METHOD Init
VAR_INPUT
  pMsgConfig : POINTER TO ST_MSG_CONFIG;         // message config
  fPrintResolution : LREAL := 1;                 // print(head) resolution in [dpi]
  fSubPxResolution : LREAL := 1;                 // SubPixel resolution [SubPx], resolution factor (fI_PrintResolution*fI_SubPxResolution=>Output resolution)
  bParallelCT : BOOL;                            // Support parallel processing of CTs
END_VAR
SUPER^.Init(pMsgConfig:=pMsgConfig, fPrintResolution:=fPrintResolution, fSubPxResolution:=fSubPxResolution, bParallelCT:=bParallelCT);

// Init messages
fbMsg_PythonNotRunning.pI_MsgConfig := _pMsgConfigExt;
fbMsg_PythonNotRunning.iI_MsgLocation := TO_INT(ePr_BLK_PU);
fbMsg_PythonNotRunning.iI_MsgNumber := eC_STAG_DEF_SCRIPT_NOT_RUNNING;
END_METHOD

METHOD InitWorkerPython
VAR_INPUT
  aScriptPath : T_MaxString;                     // path to cmd scripts
  //aAmsLocalHost : T_AmsNetID;                    // Ams netId localhost of the pc to run the script
  iDefGridParamMediator : I_ParamMediator;
END_VAR
IF NOT bInitialized OR _pCTM = 0 THEN LogError('Base Worker not initialized! call init() before'); RETURN; END_IF
IF iDefGridParamMediator = 0 THEN bInitialized := FALSE; LogError('Invalid parameter, no valid param mediator'); RETURN; END_IF

// worker specific init
_iParamMediator := iDefGridParamMediator;

fbPythonInterface.Init(
  sCTManagerPath := _pCTM^.sCTDefGridInstancesPath, 
  sScriptPath:=aScriptPath
);
END_METHOD

METHOD mJobStart
VAR_INPUT
	sJobDef	: CalmarCompPrint.I_JobDefinition;
END_VAR
// checks and fix defaults
IF _iParamMediator = 0 THEN LogError('JobStart: invalid parameter configuration'); RETURN; END_IF
IF _fWorkerPosition = 0 THEN _fWorkerPosition := fC_DEFAULT_WOKER_POSITION; LogError(F_Concat3(_name, ': worker position not set, set default=', TO_STRING(fC_DEFAULT_WOKER_POSITION))); END_IF

// configure
_aJobName := sJobDef.aJobName;
_aJobGuid := sJobDef.aJobId;
_fImageDepthM := sJobDef.fImageDepth/1000;
_fImageWidthM := sJobDef.fImageWidth/1000;

_bNewJob := TRUE;
_bJobActive := TRUE;
END_METHOD

METHOD  mJobStop
VAR_INPUT
	sStatus	: CalmarCompPrint.I_JobStatus;
END_VAR
fbPythonInterface.JobStop();
_bJobActive := FALSE;
END_METHOD

METHOD  work
VAR_INPUT
END_VAR
VAR
  i : UDINT;
  tempCt  : POINTER TO FB_ContainerDefGrid;
  bDeformationDone : BOOL;
  bDeformationError : BOOL;
END_VAR
VAR_INST
  rT_EnablePyIf  : R_TRIG;
END_VAR
SUPER^.work();

IF _iParamMediator = 0 THEN F_Report_Error(ErrType:=EN_REPORT_ERROR_TYPE.Report_Error_0Pointer); RETURN; END_IF
_CamGridSettings := _iParamMediator.sCameraGridSettings;
_DefGridSettings := _iParamMediator.sDeformationGridSettings;

// reconfig script after job started (Mediator parameter are defined in JobStart())
IF _bNewJob OR rT_EnablePyIf.Q THEN   // new job activated or re-enabled
  _bNewJob := FALSE;
  
  // setup script
  fbPythonInterface.JobStart(
    aJobName:=_aJobName,
    aJobGuid:=_aJobGuid,
    nJobImageWidth:=DINT_TO_UDINT(F_MeterToSubPixel(fPosMeter:=_fImageDepthM, fResoSubPx:=_fPrintResolution)),
    nJobImageHeigth:=DINT_TO_UDINT(F_MeterToSubPixel(fPosMeter:=_fImageWidthM, fResoSubPx:=_fPrintResolution)),
    nCamFrameWidth:=DINT_TO_UDINT(FC_LREAL_TO_DINT(_CamGridSettings.fGridFeaturePitch)),
    pGridSettings:=ADR(_DefGridSettings)
  );
END_IF

// start/stop script
IF _CamGridSettings.eCameraMode >= E_CameraMode.Live AND THIS^.bWorkerEnable THEN 
  fbPythonInterface.bEnable := TRUE;
ELSE
  fbPythonInterface.bEnable := FALSE;
END_IF
rT_EnablePyIf(CLK:=fbPythonInterface.bEnable);

fbPythonInterface();

IF _pAttachedCt <> 0 THEN
  // nothing to do anymore just release CT
  // NOTE: the delete of the CT is done by DeleteDefCt() method directly into fbPythonInterface
  Release(_pAttachedCt^);
END_IF

// messages
fbMsg_PythonNotRunning(bI_Status:=fbPythonInterface.bError);
IF fbMsg_PythonNotRunning.bMsgAck THEN fbPythonInterface.ackError(); END_IF
END_METHOD

END_FUNCTION_BLOCK

// ---- POUs/Print/DefGrid/FB_WorkerDefGrid_Verify.TcPOU
FUNCTION_BLOCK FB_WorkerDefGrid_Verify EXTENDS FB_WorkerDefGrid
VAR_OUTPUT
  bWateGateActive   AT%Q* : BOOL;     //  wate gate activation pulse
END_VAR
VAR
  bLastEject   : BOOL;   // stores state if last CT TRUE:=Eject, FALSE:=OK
  tpEjectPulse  : TP := (PT:=T#80MS);
  
  // print manager reference
  _pPm : POINTER TO FB_ProdManager_DMAX;
  
  // view verify history
  tpShowResult : TP := (PT:=T#700MS);
  nStateHistory : ARRAY[1..20] OF UINT;   // 2=???, 1=Eject, 0=OK
  nStateHistory_FillColor : ARRAY[1..20] OF UDINT;
  sResultText : STRING;
  
  // Grid Table export
  nCTId : DINT;
  bEnableGridExport : BOOL;
  nExportWrites : UDINT;
  sOutputPath : T_MaxString := 'C:\GridExport';
  sFileFormat : STRING := 'json';
  fbGridExporter : FB_GridDataExporter;
END_VAR

METHOD PROTECTED  Attach : BOOL
VAR_INPUT
  iCT              : I_CT;                         (*container at triggered event position*)
END_VAR
VAR 
  bSuccess         : BOOL;
END_VAR
IF SUPER^.Attach(iCT:=iCT) THEN
  
  // do CT supervision here and decice what happens with this sheet
   bSuccess := TRUE;
  IF NOT iCT.bValid AND iCT.bProductPresent AND iCT.pJob <> 0 THEN
    bSuccess := FALSE;
    // tag for ejection
    iCT.pCT^.lPrOutput := EN_PrinterOutput.trash;
	END_IF

  // finish CT in production
  IF _pPm <> 0 THEN 
    _pPm^.CT_Finish(sCT:=iCT, bSuccess:=bSuccess);      // report to job status
  ELSE
    LogError('PrintManager not set');
	END_IF
  
  // select output
  IF iCT.pCT^.lPrOutput = EN_PrinterOutput.trash THEN
    // create eject trigger
    tpEjectPulse(IN:=TRUE);
    bLastEject := TRUE;
    LogLvl(Lvl:=E_LogSeverity.Debug, Msg:=F_Concat2('Eject CT: ', _pAttachedCt^.print(0)));
  ELSE
    tpEjectPulse(IN:=FALSE);
    bLastEject := FALSE;
	END_IF
  
  // History view
  MEMMOVE(destAddr:=ADR(nStateHistory[1+1]),           srcAddr:=ADR(nStateHistory[1]),           n:=((SIZEOF(nStateHistory)/SIZEOF(nStateHistory[1]))-1)*SIZEOF(nStateHistory[1]));
  MEMMOVE(destAddr:=ADR(nStateHistory_FillColor[1+1]), srcAddr:=ADR(nStateHistory_FillColor[1]), n:=((SIZEOF(nStateHistory_FillColor)/SIZEOF(nStateHistory_FillColor[1]))-1)*SIZEOF(nStateHistory_FillColor[1]));
  
  nStateHistory[1] := SEL(bLastEject=TRUE, 0, 1);
  sResultText := SEL(bLastEject=TRUE, 'OK', 'NOK');

  IF iCT.bProductPresent AND iCT.bValid THEN        nStateHistory_FillColor[1] := 16#FF000000 OR WebColors.LightGreen.lCode;
  ELSIF iCT.bProductPresent AND NOT iCT.bValid AND iCT.pCT^.lPrOutput = EN_PrinterOutput.trash THEN nStateHistory_FillColor[1] := 16#FF000000 OR WebColors.LightSalmon.lCode;   
  ELSIF iCT.bProductPresent AND NOT iCT.bValid AND iCT.pCT^.lPrOutput <> EN_PrinterOutput.trash THEN nStateHistory_FillColor[1] := 16#FF000000 OR WebColors.LightGray.lCode;
	ELSIF NOT iCT.bProductPresent THEN                nStateHistory_FillColor[1] := 16#FF000000 OR WebColors.LightGray.lCode;
  END_IF

  tpShowResult(IN:=FALSE);
  tpShowResult(IN:=TRUE);
  
  // grid history
  IF bEnableGridExport AND iCT.bProductPresent AND nExportWrites < 100 THEN
    nCTId := _pAttachedCt^.pCT^.iId;
    sFileFormat := SEL(sFileFormat='csv', 'json', 'csv');
    fbGridExporter(
        sOutputDir:=sOutputPath,
        sFileName:=F_Concat4('\Export_', TO_STRING(nCTId), '.', sFileFormat),
        pFbImageDeformation:=_pAttachedCt^.pImageDeformation,
        //nSelectGrid:=
    );
    fbGridExporter.startExport();
    nExportWrites:=nExportWrites+1;
  ELSE
    nExportWrites := 0; bEnableGridExport := FALSE;
  END_IF
END_IF
END_METHOD

(*
  Set PrintManager.
*)
METHOD InitWorkerVerify : BOOL
VAR_INPUT
  pPm : POINTER TO FB_ProdManager_DMAX;
END_VAR
IF pPm = 0 THEN LogError('Invalid Pm given'); END_IF

_pPm := pPm;  // register print manager reference
END_METHOD

METHOD   mJobStart
VAR_INPUT
	sJobDef	: CalmarCompPrint.I_JobDefinition;
END_VAR
END_METHOD

METHOD  mJobStop
VAR_INPUT
	sStatus	: CalmarCompPrint.I_JobStatus;
END_VAR
END_METHOD

METHOD Release : BOOL
VAR_INPUT
  iCT              : I_CT;                         (*container at triggered event position*)
END_VAR
IF SUPER^.Release(iCT := iCT) THEN
  ;
END_IF
END_METHOD

METHOD  work
VAR_INST
  fT_Pulse  : F_TRIG;
END_VAR
SUPER^.work();

// output signal handling
tpEjectPulse(Q=>bWateGateActive);
fT_Pulse(CLK:=bWateGateActive);
tpShowResult();
//IF tpShowResult.IN:=TRUE AND NOT tpShowResult.Q THEN tpShowResult(IN:=FALSE); END_IF   // reset pulse

fbGridExporter();

// release
IF tpEjectPulse.IN THEN
  IF fT_Pulse.Q THEN  
    tpEjectPulse(IN:=FALSE);
  END_IF
END_IF

IF _pAttachedCt <> 0 THEN   // just release any attached container in this cycle
  Release(iCT:=_pAttachedCt^);
END_IF
END_METHOD

END_FUNCTION_BLOCK

// ---- POUs/Print/Maxliner/FB_PrintModule_Maxliner.TcPOU
(*
  A DVT PrintModule (DEU, DSU, WEU).
*)
FUNCTION_BLOCK FB_PrintModule_Maxliner EXTENDS T_NamedBase IMPLEMENTS I_Sim, I_PositionEvent
VAR_INPUT
  // encoder input --> directly mapped into FB_PrintPosition 
  // machine state by pointer in init()
  // external start pos interface by pointer in init()
  fPrintOffsetX           : LREAL;   // [m] external configurative offsets to PM (PU)
  fPrintOffsetY           : LREAL;   // [m] external configurative offsets to PM (PU)

  fPUPlate1_Temperature   : LREAL;  // PU Plate1 temperature
END_VAR

VAR
  //config

  // - references
  _pModuleSetup           : POINTER TO ST_CassetteSetup;
  _iPrintGlobal           : I_PrintGlobal;        // master module (setting, position, global stuff, ...)
  _iPrintPosition         : I_PrintPosition;      // module's position
  _iStartPos              : I_StartPosDetect;     // module's start position detect
  _iModule                : I_Module;             // module's system status
  _pModuleMachineState    : POINTER TO ST_ModuleMachineInterface_IN;   // machine interface-print states
  _pModuleMachineFeedback : POINTER TO ST_ModuleMachineInterface_OUT;  // machine interface-print feedback
    
  // status
  bInit                   : BOOL;   // initialized
  bSelectedForPrint       : BOOL;   // selected for printing
  bReadyForPrinting       : BOOL;   // Module ready for printing
  bHardwareHold           : BOOL;   // hw hold
  _bGridLimited           : BOOL;   // calculated grid was limited before sending
  
  // instances
  fbPrintPosition         : FB_PrintPositionDmax;   // a position per pm (external encoder wheel)

  fbCTTracker             : FB_CTTracker;
  fbParamMediator         : FB_DefGridParamMediator;
  fbWorkerPython          : FB_WorkerDefGrid_Python;
  fbWorkerCamera          : FB_WorkerDefGrid_Camera;
  fbWorkerDeformation     : FB_WorkerDefGrid_Deformation;
  fbWorkerPrint           : ARRAY[1..GVL_Maxliner.nC_MaxWorkerPrintPerPm] OF FB_WorkerDefGrid_Print;
  
  _pAdsSa                 : POINTER TO FB_ADS_DVTSHEETALIGNMENT; // sheet alignement ads
  fbAdsPm                 : FB_ADS_PM;      // PM -  Print Module ADS
  fbAdsPg                 : ARRAY[1..GVL_Maxliner.nC_MaxWorkerPrintPerPm] OF FB_ADS_PG;  // PG - PrintGroup ADS
  
  // hw (references only for now) ------
  // - pc
  _pPc                    : ARRAY[1..GVL_Maxliner.nC_MaxPcPerPm] OF POINTER TO FB_PC;
  _nPc                    : UDINT;  // number of PC in module
  _nPcToWorker_Mapping    : ARRAY[1..GVL_Maxliner.nC_MaxPcPerPm] OF UDINT;   // Mapping of PC to worker  
  _nPcToPgAbsoluteIdx     : ARRAY[1..GVL_Maxliner.nC_MaxPcPerPm] OF UDINT;   // Mapping of PC to absolute PG index
  // - ph
  _pPh                    : ARRAY[1..GVL_Maxliner.nC_MaxPhPerPm] OF POINTER TO FB_PH;
  _nPh                    : UDINT;  // number of PH in module
  _nPhToWorker_Mapping    : ARRAY[1..GVL_Maxliner.nC_MaxPhPerPm] OF UDINT;  // Mapping of PH to worker
  _nPhToPc_Mapping        : ARRAY[1..GVL_Maxliner.nC_MaxPhPerPm] OF UDINT;  // Mapping of PH to PC
  _nPhToPcCh_Mapping      : ARRAY[1..GVL_Maxliner.nC_MaxPhPerPm] OF UDINT;  // Mapping of PH to PC channel
  _nPhToPgAbsoluteIdx     : ARRAY[1..GVL_Maxliner.nC_MaxPhPerPm] OF UDINT;  // Mapping of PH to absolute PG index
  
  // helper
  nCtr                    : UDINT;
  nYShift_PcRamCenter     : UDINT;     // y-shift for centered image in CB RAM [px]
  fSpeed, fSpeedMpMin     : LREAL;
  bSpeedReachedForPrinting: BOOL;      // Speed for printing reached
  nPos_SubPx, nPos_Px     : DINT;
  nPos_SubPx_mem          : DINT;
  fPos_um                 : LREAL;
  nTrackPosMain           : DINT;      // tracker attach position - module position relative to pos reference in main tracker [m]

  bHwSyncCmd              : BOOL;
  sCamGridSettings        : ST_CameraGridSettings;
  bOnePgActive            : BOOL;

  // sync CT trigger with Camera detection
  _bNewCT                 : BOOL;   // a new ct is received to be treated
  _iNewCT                 : I_CT;   // new ct to be treated
  _bNewStartPosX0         : BOOL;   // a new startpos detected by cam
  _nNewStartPosX0         : DINT;   // new startpos X0 deteced by cam

  fbFineAlignement        : FB_FineAlignement;     // additional grid corrections, PU Deformation/correction (4p, banana, ...)

  // messaging
  fb_MsgQueue             : FB_MSG_QUEUE;                 (*Message queue*)
  fb_MsgHandler           : FB_MSG_HANDLER;               (*Message handler*)
  sL_MsgConfig            : ST_MSG_CONFIG;                (*Message config*)
//fbMsg                   : ARRAY [1..nC_NumMsg] OF FB_MESSAGE;  (*Messages*)
  
  // simulation
  fbSim                   : FB_Sim;

  // view
  fbView                  : FB_PrintModule_Maxliner_View;    // additional controls for print module visus

  // test
  bTestMsg : BOOL;      // activate message test
END_VAR

VAR PERSISTENT
  _fPmDistToPrev          : LREAL;                 // [m] distance to previous PM (in main domain)
  _fPmMainTrackPos        : LREAL;                 // [m] used distance to master reference position (in main tracker)
END_VAR

VAR CONSTANT
  nC_NumMsg               : UDINT := 0;            // number of internal messages
  fC_HeadOffsetPlate      : LREAL := 0.000_2;      // Head offset to base plate [m] (mechanical)
  fC_MinimalProductionSpeed_in_MpMin: LREAL := 5.0;    // [m/min]
  fC_FormatLengthTolerance : LREAL := 100.0;       // [px] tolerance of substrate length job - machine config 
  nC_StopReadyTimeout     : TIME := T#10S;         // Synced stopping of printing, max. timeout to wait for printing end
END_VAR

IF NOT bInit THEN RETURN; END_IF

// position
fbPrintPosition.fEnoderResolution := _pModuleMachineState^.fEncoderResolution;    // encoder resolution from machine
fbPrintPosition();

// -------------------------
// StartTrigger evaluation -> apply new CT to Tracking (created from CTM externally)
// Synchronize CT (EvPos) received from CTManger (Main) to the local StartTrigger detection and positioning
// -- reset triggers if not active
IF NOT bReadyForPrinting THEN
  _bNewCT := 0; _bNewStartPosX0 := 0;
END_IF
// -- new StartTrigger (X0)
IF bReadyForPrinting AND _iStartPos.bStartTrig AND _iStartPos.bValid THEN
  // buffer/save new start trigger
  _bNewStartPosX0 := TRUE;
  _nNewStartPosX0 := _iStartPos.nStartPositionX0;      // save detected start position for next CT to be applied to this module¨
  
  LogLvl(Lvl:=E_LogSeverity.Debug, Msg:=F_Concat3(
    F_Concat2(_pModuleSetup^.aName, ' New StartTrigger detected:'),
    F_Concat2(' at position X0:', TO_STRING(_nNewStartPosX0)),
    F_Concat2(' PM is now at: ', TO_STRING(fbPrintPosition.getPosition())),
  ));
  
  IF _bNewCT THEN   // we have an attached CT
      LogLvl(Lvl:=E_LogSeverity.Debug, Msg:=F_Concat3(
      F_Concat2(_pModuleSetup^.aName, ' Track NewCT:'),
      F_Concat2(' internal (print)Pos X0:', TO_STRING(_nNewStartPosX0)),
      F_Concat2(' with CT:', _iNewCT.print(0))
    ));
    
    _iNewCT.nPosPrint_X0 := _nNewStartPosX0;                            // set print pos to new dected in this module position domain
    fbCTTracker.RegisterCT(iCT := _iNewCT, nX0 := _nNewStartPosX0);     // register ct for tracking in modules position and tracking system
  ELSE
    // spurious trigger (CTs not yet arrived at PMx, but receive some StartTriggers
    LogLvl(Lvl:=E_LogSeverity.Debug, Msg:=F_Concat3('StartTrigger at Pos X0:', TO_STRING(_nNewStartPosX0), ' but no CT received'));
	END_IF
  
  // reset internals (saved triggers)
  _bNewCT := FALSE; _iNewCT := 0; 
  _bNewStartPosX0 := FALSE;
END_IF

// positioning
// - get position 
nPos_SubPx := _iPrintPosition.getPosition(nPosition_px=>nPos_Px, fPosition_um=>fPos_um);
// (disabled) nPos_SubPx := nPos_SubPx_mem := SEL(bReadyForPrinting AND _iPrintPosition.bMoving, nPos_SubPx_mem, nPos_SubPx);   // security measure (jetting when not really moving or not in position
// - get speed
fSpeed := _iPrintPosition.getSpeed(fSpeedMpMin=>fSpeedMpMin);

// update distance from machine
_fPmDistToPrev := _pModuleMachineState^.fDistanceToPrevModule;

// enable, control, release signals
//   engaged -> selected and prepared for production
//   printActivated -> machine & axis position ready for printing
//   InitInPrintPosition -> module in pos to allow printing
bSelectedForPrint        := fbAdsPm.bEnable AND _pModuleMachineState^.bEngaged;
bSpeedReachedForPrinting := (fSpeedMpMin >= fC_MinimalProductionSpeed_in_MpMin);
// ready for printing (enable detection)
bReadyForPrinting        :=      bSelectedForPrint                                // selected and ready for production (from machine)
                            AND _pModuleMachineState^.bPrintActivated             // machine & axis ready for printing
                            AND _pModuleMachineState^.bUnitInPrintPosition        // module in printing position -> allowed to print
                            AND bSpeedReachedForPrinting                          // speed bigger than min speed for printing
                            AND _pModuleMachineState^.bTargetSpeedReached         // do not evaluate marks while machine ramping up  
                            AND NOT _pModuleMachineState^.bStopRequest            // do not evaluate marks while machine is stopping
                            AND NOT _pModuleMachineState^.bEStop
                            AND NOT _pModuleMachineState^.bSleep;
bHardwareHold            := NOT bSpeedReachedForPrinting OR 
                            NOT _pModuleMachineState^.bPrintActivated OR 
                            NOT _pModuleMachineState^.bUnitInPrintPosition OR 
                                _pModuleMachineState^.bFastStopRequest;
bHwSyncCmd               := checkHwSyncRequest();                                 // sync trigger generation

// pos for attach in main tracker
nTrackPosMain := F_MeterToSubPixel(fPosMeter:=_fPmMainTrackPos, fResoSubPx:=_iPrintPosition.fPrintResolution*_iPrintPosition.fSubPxResolution); 
// run tracker
fbCTTracker(nPos:=nPos_SubPx);


// call hardware
(* -- PC PrintController*)
FOR nCtr := 1 TO _nPc DO
  IF _pPc[nCtr] <> 0 THEN
    _pPc[nCtr]^.sI_SystemCmd.bSleep := _pModuleMachineState^.bSleep;  // from if to module (machine)
    _pPc[nCtr]^.sI_SystemCmd.bEStop := _pModuleMachineState^.bEStop;  // from if to module (machine)
    _pPc[nCtr]^.sI_SystemCmd.bAirNotOk := FALSE;
    _pPc[nCtr]^();
  END_IF
END_FOR

(* -- PH PrintHead*)
FOR nCtr := 1 TO _nPh DO
  IF _pPh[nCtr] <> 0 THEN
    ; // called in PC.update()->pPh[nCtr]^();
  END_IF
END_FOR


// Worker
// - Camera
fbWorkerCamera.bWorkerEnable := fbAdsPm.bEnable AND bOnePgActive;
sCamGridSettings := fbWorkerCamera.sCameraGridSettings;
// - Deformation
fbWorkerDeformation.bWorkerEnable := fbAdsPm.bEnable AND bOnePgActive AND sCamGridSettings.eDeformationType > E_DeformationType.NoDeformation;

// - Print
// - fill I_SubSystem correctly from all workers
FOR nCtr := 1 TO GVL_Maxliner.nC_MaxWorkerPrintPerPm DO
  fbWorkerPrint[nCtr].bWorkerEnable := fbAdsPm.bEnable AND fbWorkerPrint[nCtr]._pAdsPg^.bEnable;
  //fbWorkerPrint[nCtr].bWorkerPrintEnable := _pModuleMachineState^.bPrintActivated;
  fbWorkerPrint[nCtr](
    nEncoderPos           := nPos_SubPx,
    fMasterSpeed          := fSpeed,
    bHardwareSync         := bHwSyncCmd,
    bHardwareHold         := bHardwareHold,
  //nPhDepth              := _pModuleSetup^.pSetupPrint^.sPHType.iC_Ph_Depth,
  //bFastStopRequest      := _pModuleMachineState^.bFastStopRequest,
  //bPrintStopRequest     := _pModuleMachineState^.bStopRequest,
                            // Print StartPosition Distance to detected X0 of CT
    fPrintStartOffset     :=   fPrintOffsetX                                    // NOTE: dynamic corrections done in Worker (dropSpeedComp / global grid dx / other point corrections))
                             - TO_LREAL(fbAdsPm.nGeneralShiftX) / 1_000_000     // ! negative direction to match PUC UI => change requested by STAG (14.08.2024)
                             + TO_LREAL(fbAdsPg[nCtr].nPositionX) / 1_000_000,
    fPrintYOffset         := LIMIT(
                              0,
                                F_SubPixelToMeter(TO_DINT(nYShift_PcRamCenter), _iPrintPosition.fPrintResolution)              // y-offset for centered image in ph
                                + fPrintOffsetY
                                - TO_LREAL(fbAdsPm.nGeneralShiftY) / 1_000_000    // ! negative direction to match PUC UI => change requested by STAG (16.12.2024)
                                + TO_LREAL(fbAdsPg[nCtr].nPositionY) / 1_000_000
                                + _pModuleMachineState^.fLateralRegister  // lateral register from machine
                              ,2*F_SubPixelToMeter(TO_DINT(nYShift_PcRamCenter), _iPrintPosition.fPrintResolution)
                            ),
    fPUElevation          := _pModuleMachineFeedback^.fHeadGap, // + fC_HeadOffsetPlate,
//    bError                => ,
//    nError                => ,
  );
END_FOR

// collect printWorker status
FOR nCtr := 1 TO GVL_Maxliner.nC_MaxWorkerPrintPerPm DO
  IF fbWorkerPrint[nCtr].bWorkerEnable THEN
    _bGridLimited := fbWorkerPrint[nCtr]._bGridWasLimited OR _bGridLimited; 
	END_IF
END_FOR

// One PG (printWorker) active
bOnePgActive := FALSE;
FOR nCtr := 1 TO GVL_Maxliner.nC_MaxWorkerPrintPerPm DO 
  IF fbAdsPg[nCtr].bEnable THEN bOnePgActive := TRUE; END_IF 
END_FOR

  
// machine interface outputs
_pModuleMachineFeedback^.bMoving           := bSpeedReachedForPrinting;
_pModuleMachineFeedback^.fSpeed            := fSpeed;
_pModuleMachineFeedback^.fPosition         := fPos_um / 1_000_000;
_pModuleMachineFeedback^.bSpeedExeeded     := checkSpeed(fSpeed:=fSpeed, fMaxSpeed => _pModuleMachineFeedback^.fMaxSpeed);
_pModuleMachineFeedback^.bLengthMismatch   := checkFormatLength();
_pModuleMachineFeedback^.bStopReady        := checkReadyForStop(bStopRequestSync:=_pModuleMachineState^.bStopRequest);
_pModuleMachineFeedback^.fHeadGap          := _pAdsSa^.fHeadGap / 1000;  // [mm] -> [m]
_pModuleMachineFeedback^.fInkQuantity      := getInkQuantity();

(*PU corrections*)
IF GVL_Deformation.bC_UsePUDeformation THEN
  fbFineAlignement.fT_PL1 := fPUPlate1_Temperature;
  fbFineAlignement.fT_PL2 := fPUPlate1_Temperature;  // Plate2 not existing
  fbFineAlignement();
END_IF

// simulation
SimUpdate();

// view
fbView();

// messaging
Messaging();

{attribute 'monitoring':='call'}
PROPERTY bMoving : BOOL
GET
bMoving := _iPrintPosition.bMoving;
END_GET
END_PROPERTY

{attribute 'monitoring' := 'call'}
// module is selected for production (and considered in positioning)
PROPERTY bSelectedForProduction : BOOL
GET
bSelectedForProduction := bSelectedForPrint;
END_GET
END_PROPERTY

{attribute 'monitoring' := 'call'}
(*Simulation is enabled set/get*)
PROPERTY bSimEnable : BOOL
GET
bSimEnable := fbSim.bSimEnable;
END_GET
SET
fbSim.bSimEnable := bSimEnable;
END_SET
END_PROPERTY

(* 
  Hardware sync request.
*)
PROPERTY bSyncCmd : BOOL
GET
bSyncCmd := bHwSyncCmd;
END_GET
END_PROPERTY

// check imagelength vs formatlength
// :returns: TRUE if a mismatch was detected
METHOD PRIVATE checkFormatLength : BOOL
VAR 
  nFormatTolerance : LREAL;
  bOneJobActive    : BOOL;
  i                : UDINT;
  _fImageLength    : LREAL;
END_VAR
// check config
_fImageLength := 0;
FOR i := 1 TO GVL_Maxliner.nC_MaxWorkerPrintPerPm DO
  IF fbWorkerPrint[i]._bEnable THEN
    _fImageLength := fbWorkerPrint[i].fImageLength;
	END_IF
END_FOR

IF _fImageLength = 0 THEN RETURN; END_IF
IF _pModuleMachineState^.fSubstrateLen = 0 THEN RETURN; END_IF
IF bSimEnable THEN RETURN; END_IF  // check ok during simulation

bOneJobActive := FALSE;
FOR i := 1 TO GVL_Maxliner.nC_MaxWorkerPrintPerPm DO
  bOneJobActive := bOneJobActive OR fbWorkerPrint[i].bJobActive;
END_FOR
IF NOT bOneJobActive THEN RETURN; END_IF

// compare
nFormatTolerance := fC_FormatLengthTolerance / _pModuleSetup^.pSetupPrint^.nPrintResolution * 0.0254;  // 100 [px] -> [m]
IF nFormatTolerance < ABS(_fImageLength - _pModuleMachineState^.fSubstrateLen) THEN
  checkFormatLength := TRUE;
END_IF
END_METHOD

METHOD PROTECTED checkHwSyncRequest : BOOL
VAR_INST
  rT_SyncRequest : R_TRIG;
  tSyncDelay     : TON;
END_VAR
VAR_OUTPUT
  bHwSyncReq : BOOL;
END_VAR
rT_SyncRequest(CLK:=bReadyForPrinting);
IF rT_SyncRequest.Q OR _iPrintPosition.bStarted THEN  // OR rT_JobActive.Q 
  tSyncDelay(IN:=TRUE, PT:=T#2MS);   // a Sync delay to workaround a sync sent to CB while a Start or Prepare Command
END_IF
tSyncDelay(Q=>bHwSyncReq);
IF tSyncDelay.Q THEN 
  tSyncDelay(IN:=FALSE);
END_IF


checkHwSyncRequest := bHwSyncReq;
END_METHOD

METHOD PRIVATE checkReadyForStop : BOOL
VAR_INPUT
  bStopRequestSync : BOOL;
END_VAR
VAR
  i : UDINT;
  bStopReady : BOOL;
END_VAR
VAR_INST
  tOnStoppingSupversion : TON;  // check if it takes too long for stopping print with (synced)stop-request
  rTSupervsion : R_TRIG;
END_VAR
// check print states
bStopReady := TRUE;
FOR i := 1 TO GVL_Maxliner.nC_MaxWorkerPrintPerPm DO                        // all worker stopped?
  bStopReady := bStopReady AND NOT fbWorkerPrint[i].bPrintActive;   // stop ready if no print is active
END_FOR

// error handling
// - 
tOnStoppingSupversion(IN:=bStopRequestSync AND NOT bStopReady, PT:=nC_StopReadyTimeout);   // supervision for synchronized stopping the print of module
rTSupervsion(CLK:=bStopRequestSync AND tOnStoppingSupversion.Q);    // 
IF rTSupervsion.Q THEN LogWarning('checkReadyForStop: stopped by timeout (stop ready not received from PM)'); END_IF


// ready if request set and all finished printing (or supervision)
checkReadyForStop := bStopRequestSync AND (bStopReady OR tOnStoppingSupversion.Q);
END_METHOD

(*
  Checks if current speed is higher than max. speed.
  :return: TRUE if speed exeeds maximum
*)
METHOD PROTECTED checkSpeed : BOOL
VAR_INPUT
  fSpeed : LREAL;       // current speed
END_VAR
VAR_OUTPUT
  fMaxSpeed : LREAL;    // modules max. printing speed
END_VAR
VAR
  f : LREAL;
  i : UDINT;
END_VAR
VAR_INST
  fbSpeedFilterMav : FB_FILTER_MAV;           // Moving average filter
  fMaxSpeedTolerence : LREAL := 1.0/60;       // Allow max. speed to exeed limit + this tolerance 
END_VAR
// disabled
IF NOT fbAdsPm.bEnable OR NOT _pModuleMachineState^.bEngaged THEN 
  checkSpeed := FALSE;
  fMaxSpeed := 0;
  RETURN;
END_IF 


// filter current speed
fbSpeedFilterMav(fI_Input := fSpeed, iI_NbInputs := 32);  (*max iI_NbInputs = 32!*)

// find slowest max. speed
f := 0;
FOR i:=1 TO GVL_Maxliner.nC_MaxWorkerPrintPerPm DO
  IF fbWorkerPrint[i].bWorkerEnable THEN
    IF fbWorkerPrint[i].fMaxSpeed = 0 THEN
      ; // ignored speed
    ELSIF f = 0 OR f > fbWorkerPrint[i].fMaxSpeed THEN 
      f := fbWorkerPrint[i].fMaxSpeed;
		END_IF
	END_IF
END_FOR

fMaxSpeed := f;   // return max. possible speed

// check if too fast
IF f > 0 AND fbSpeedFilterMav.fO_OutputMav > (f+fMaxSpeedTolerence) THEN 
  checkSpeed := TRUE; // speed exceeded
ELSE
  checkSpeed := FALSE;
END_IF
END_METHOD

(*
  Distance between activated StartPosition detection and Pm, if one configured (fDetectToCameraOffset + fCameraToPrintOffset)
  If no StartPos detection = 0
*)
PROPERTY fDetectToPm : LREAL
GET
fDetectToPm := fbWorkerCamera.fDetectToCamOffset + fbWorkerCamera.fCameraToPrintOffset;
END_GET
END_PROPERTY

// distance to previous print module (on master tracking pos)
PROPERTY fPmDistToPrev : LREAL
GET
fPmDistToPrev := _fPmDistToPrev;
END_GET
SET
_fPmDistToPrev := fPmDistToPrev;
END_SET
END_PROPERTY

PROPERTY fPmMainTrackPos : LREAL
GET
fPmMainTrackPos := _fPmMainTrackPos;
END_GET
SET
_fPmMainTrackPos := fPmMainTrackPos;
END_SET
END_PROPERTY

METHOD getInkQuantity : LREAL
VAR
  nWorker : UDINT;
END_VAR
FOR nWorker := 1 TO GVL_Maxliner.nC_MaxWorkerPrintPerPm DO
  IF fbWorkerPrint[nWorker].bWorkerEnable THEN    // from first enabled worker (PG)
    getInkQuantity := fbWorkerPrint[nWorker]._pAdsPg^.lInkQuantity;
    EXIT;
	END_IF
END_FOR
END_METHOD

METHOD Init : BOOL
VAR_INPUT
  pModulesSetup         : POINTER TO ST_CassetteSetup;          // Module Setup Settings
  pAdsSa                : POINTER TO FB_ADS_DVTSHEETALIGNMENT;  // ADS sheet alignement
  pAdsCam               : POINTER TO FB_ADS_CAMERA;             // ADS camera
  pAdsParent            : POINTER TO FB_ADS_Config;             // Parent ADS config reference (Parent ADS block and module ref)

  // config print
  fCycleTime            : LREAL;                // task cycle time in [s]
  fPrintUnitWidth       : LREAL;                // PrintUnit width mechanical [m]
  // references
  iModule               : I_Module;             // system status interface (for sleep, estop, ...), may shadow states from machine inputs
  iPrintGlobal          : I_PrintGlobal;        // interface for module to master (main) communication
  pMachineInputs        : POINTER TO ST_ModuleMachineInterface_IN;
  pMachineOutputs       : POINTER TO ST_ModuleMachineInterface_OUT;

  iStartPos             : I_StartPosDetect;     // module's start position detect
END_VAR

VAR
  nCtr : UDINT;
  sMode : ST_SimModeDef;
END_VAR
IF         pModulesSetup = 0 
   OR_ELSE pAdsSa = 0 
   OR_ELSE pAdsCam = 0 
   OR_ELSE pAdsParent = 0 
   OR_ELSE pMachineInputs = 0 
   OR_ELSE pMachineOutputs = 0 
   OR_ELSE iPrintGlobal = 0 
THEN
  LogError('init(): Invalid parameter');
  RETURN;
END_IF

// save config
_pModuleSetup := pModulesSetup;
_pAdsSa := pAdsSa;
_iPrintGlobal := iPrintGlobal;
_iModule := iModule;
_pModuleMachineState := pMachineInputs;
_pModuleMachineFeedback := pMachineOutputs;
nYShift_PcRamCenter := _pModuleSetup^.pSetupPrint^.nPcYShiftCenterRam;

// -- Sheet/Camera
_iStartPos := iStartPos;  // select start position detection


// init & setup hw and module linking
SetupHw();

// ADS config and mapping
InitAds(pAdsParent:=pAdsParent);

// position
fbPrintPosition.Init(fPrintResolution := pModulesSetup^.pSetupPrint^.nPrintResolution, fSubPxResolution := pModulesSetup^.pSetupPrint^.nSubPixelResolution, fTaskCycleTime := fCycleTime);
_iPrintPosition := fbPrintPosition;  // select reference position

// cttracker
fbCTTracker.Init(aName:=F_Concat2('Tracker of ', pModulesSetup^.aName), aUnit:='SubPx', bAutoRemoveAfterLastEvPos:=TRUE);

// Worker
// -- parameter mediator
fbParamMediator.init(pCamWorker:=ADR(fbWorkerCamera), pDefWorker:=ADR(fbWorkerDeformation));

// -- Worker Python
fbWorkerPython.Init(pMsgConfig:=ADR(sL_MsgConfig), fPrintResolution:=_iPrintPosition.fPrintResolution, fSubPxResolution:=_iPrintPosition.fSubPxResolution, bParallelCT:=TRUE);
fbWorkerPython.InitWorkerPython(aScriptPath:=F_Concat2(GVL_Maxliner.aC_PlcProjectCfgPath, 'Tools\Deformation\'), iDefGridParamMediator:=fbParamMediator);
fbWorkerPython.reg();
fbCTTracker.RegisterTrackPos(iPositionEvent := fbWorkerPython);
iPrintGlobal.registerPuStatusClient(sClient := fbWorkerPython);

// -- Worker camera
fbWorkerCamera.Init(pMsgConfig:=ADR(sL_MsgConfig), fPrintResolution:=_iPrintPosition.fPrintResolution, fSubPxResolution:=_iPrintPosition.fSubPxResolution, bParallelCT:=TRUE);
fbWorkerCamera.InitWorkerCamera(pAdsIf:=pAdsCam, iDefGridParamMediator:=fbParamMediator, fFeatureGrid:=256, fPrintUnitWidth:=fPrintUnitWidth);
fbWorkerCamera.reg();
fbCTTracker.RegisterTrackPos(iPositionEvent := fbWorkerCamera);
iPrintGlobal.registerPuStatusClient(sClient := fbWorkerCamera);

// -- Worker deformation
fbWorkerDeformation.Init(pMsgConfig:=ADR(sL_MsgConfig), fPrintResolution:=_iPrintPosition.fPrintResolution, fSubPxResolution:=_iPrintPosition.fSubPxResolution, bParallelCT:=TRUE);
fbWorkerDeformation.InitWorkerDeformation(nPrintUnitWidth:=TO_UDINT(F_MeterToSubPixel(fPosMeter:=fPrintUnitWidth, fResoSubPx:=_iPrintPosition.fPrintResolution)), iDefGridParamMediator:=fbParamMediator);
fbWorkerDeformation.reg();
fbCTTracker.RegisterTrackPos(iPositionEvent := fbWorkerDeformation);
iPrintGlobal.registerPuStatusClient(sClient := fbWorkerDeformation);

// -- Worker print
FOR nCtr := 1 TO GVL_Maxliner.nC_MaxWorkerPrintPerPm DO
  fbWorkerPrint[nCtr].Init(
    fPrintResolution:=_iPrintPosition.fPrintResolution,
    fSubPxResolution:=_iPrintPosition.fSubPxResolution,
    pMsgConfig:=ADR(sL_MsgConfig),
    bParallelCT:=TRUE
  );
  fbWorkerPrint[nCtr].InitWorkerPrint(
    pAdsPg                := ADR(fbAdsPg[nCtr]),
    iDefGridParamMediator := fbParamMediator,
    fPrintUnitWidth       := fPrintUnitWidth,
    fLimitCorrectionX     := 1000,
    fLimitCorrectionY     := nYShift_PcRamCenter - 1
  );
  fbWorkerPrint[nCtr].reg();
  fbCTTracker.RegisterTrackPos(iPositionEvent := fbWorkerPrint[nCtr]);
  iPrintGlobal.registerPuSubystem(iSubSys := fbWorkerPrint[nCtr]);
END_FOR

// additional grid point corrections
fbFineAlignement.init(pAdsCam := pAdsCam, fPxReso := _iPrintPosition.fPrintResolution, fPuWidth := fPrintUnitWidth);
// - register them to workers
(*Register not existing yet
FOR nCtr := 1 TO GVL_Maxliner.nC_MaxWorkerPrintPerPm DO
  fbWorkerPrint[nCtr].RegisterGridCorrection(iGridCorrection := fbFineAlignement);
END_FOR *)

fbView.init(pModule := THIS, pPositioning := ADR(fbPrintPosition));

(*Messaging*)
sL_MsgConfig.bI_Enable       := TRUE;
sL_MsgConfig.pI_FbMsgHandler := ADR(fb_MsgHandler);
fb_MsgHandler.pI_MsgQueue    := ADR(fb_MsgQueue);
fb_MsgQueue.pI_MsgInterface  := fbAdsPm.pMsgInterface;
fb_MsgQueue.cI_MaxElement    := TO_INT(SIZEOF(fbAdsPm.pMsgInterface^.sO_MsgBuffer)/SIZEOF(ST_ADS_MSG));

(*Messages*)
(*
FOR nCtr := 1 TO nC_NumMsg DO
  fbMsg[nCtr].pI_MsgConfig   := ADR(sL_MsgConfig);
  fbMsg[nCtr].iI_MsgLocation := 1;
END_FOR;

fbMsg[ 1].iI_MsgNumber       := ;     // mark detection error
*)
Init := bInit := TRUE;
END_METHOD

// ADS Configuration of interface 
// ADS Block Mapping of Module
METHOD PROTECTED InitAds
VAR_INPUT
  pAdsParent  : POINTER TO FB_ADS_Config;             // Parent ADS config reference (Parent ADS block and module ref)
END_VAR
// ADS Mapping --------------------------------------------
// -> to PU
pAdsParent^.register(ADR(fbAdsPm));  // PM -->PU
// -> to PM
FOR nCtr := 1 TO GVL_Maxliner.nC_MaxWorkerPrintPerPm DO
  pAdsParent^.iAdsParent := fbAdsPm;
  pAdsParent^.register(ADR(fbAdsPg[nCtr]));    // PG --> PM
  (*groups -> header tank group*)
  pAdsParent^.iAdsParent := _pModuleSetup^.pSetupInk^.pInkHeaderTankGroup^;
  pAdsParent^.register(ADR(fbAdsPg[nCtr]));    // PG --> HT Group
END_FOR

// -> to PG
FOR nCtr := 1 TO _nPc DO
  pAdsParent^.iAdsParent := fbAdsPg[_nPcToWorker_Mapping[nCtr]];
  pAdsParent^.register(_pPc[nCtr]^.pAdsBlock);     // PC --> PG
END_FOR;

// -> to PC
(*printhead*)
FOR nCtr := 1 TO _nPh DO
  pAdsParent^.iAdsParent := _pPc[_nPhToPc_Mapping[nCtr]]^.pAdsBlock^;
  pAdsParent^.register(_pPh[nCtr]^.pAdsBlock);    // PH --> PC
END_FOR;


// ADS Config ---------------------------------------------
(* -- PM PrintModuile*)
fbAdsPm.aName := _pModuleSetup^.aName;
fbAdsPm.config(
    bGeneralShiftX_Exist := TRUE
  , aGeneralShiftX_Unit  :=  'um'
  , nGeneralShiftX_Min   := -380_000
  , nGeneralShiftX_Max   := 1_000_000
  
  , bGeneralShiftY_Exist := TRUE
  , aGeneralShiftY_Unit  := 'um'
  , nGeneralShiftY_Min   := -8_001
  , nGeneralShiftY_Max   := 8_001
);

(* -- PG PrintGroup*)
FOR nCtr := 1 TO GVL_Maxliner.nC_MaxWorkerPrintPerPm DO
  fbAdsPg[nCtr].aName := F_Concat4(fbAdsPm.aName, ' - ', 'Printline ', TO_STRING(nCtr));
  fbAdsPg[nCtr].config(
       bShiftPositionX_Exist     := TRUE
     , aShiftPositionX_Unit      := 'um'
     , lShiftPositionX_Min       := 0
     , lShiftPositionX_Max       := 2_000_000
     
     , bShiftPositionY_Exist     := FALSE
     , aShiftPositionY_Unit      := 'pixel'
     , lShiftPositionY_Min       := 0
     , lShiftPositionY_Max       := 2147483647
     
     , bInkQuantity_Exist        := FALSE
     , aInkQuantity_Unit         := 'g/m^2'
     , lInkQuantity_Min          := 0
     , lInkQuantity_Max          := 100
     
     , bMaxPrintSpeed_Exist      := FALSE
     , aMaxPrintSpeed_Unit       := 'm/min'
     , lMaxPrintSpeed_Min        := 0
     , lMaxPrintSpeed_Max        := 100
  );
END_FOR;
END_METHOD

PROPERTY iPrintPosition : I_PrintPosition
GET
iPrintPosition := _iPrintPosition;
END_GET
END_PROPERTY

PROPERTY iStartPos : I_StartPosDetect
GET
iStartPos := _iStartPos;
END_GET
END_PROPERTY

METHOD PRIVATE Messaging
VAR_INPUT
END_VAR
(*Messaging*)
fb_MsgHandler();
fb_MsgQueue();

// messages print module
//fbMsg[ 1](bI_Status := bTestMsg OR );

// message ack
IF fb_MsgQueue.bO_ReceiptMessage THEN
  IF bTestMsg THEN LogInfo('Ack messages'); END_IF
END_IF
END_METHOD

PROPERTY nTrackOffset : DINT
GET
nTrackOffset := nTrackPosMain;
END_GET
END_PROPERTY

(*
  NOTE: Only needed because the Hw instances are outside of the Module.
        Please call the register HW prior initializing the Module itself!
*)
METHOD RegisterHw : BOOL
VAR_INPUT
  pPh : POINTER TO FB_PH;
  pPc : POINTER TO FB_PC;
  pMapDef : POINTER TO ST_MappingDefinition;
END_VAR
VAR
  i : UDINT;
  bFound : BOOL;
END_VAR
IF pPh = 0 OR pPc = 0 OR pMapDef = 0 THEN LogError('registerHw invalid parameter'); RETURN; END_IF
IF _nPc >= GVL_Maxliner.nC_MaxPcPerPm THEN LogError('register hw: too many PCs registered'); RETURN; END_IF
IF _nPh >= GVL_Maxliner.nC_MaxPhPerPm THEN LogError('register hw: too many PHs registered'); RETURN; END_IF

// PC 
bFound := FALSE;
FOR i:=1 TO _nPc DO   // search for existing pc
  IF _pPc[i] = pPc THEN bFound := TRUE; EXIT; END_IF
END_FOR
IF NOT bFound THEN    // add if unknown
  _nPc := _nPc + 1;
  _pPc                [_nPc] := pPc;
  _nPcToWorker_Mapping[_nPc] := pMapDef^.nPg;  // save mapping
  _nPcToPgAbsoluteIdx [_nPc] := pMapDef^.nPgAbs;  // save PCs mapping to PG absolute
ELSE
  ; // ignore new pc
END_IF

// PH
bFound := FALSE;
FOR i:=1 TO _nPh DO   // search for existing ph
  IF _pPh[i] = pPh THEN bFound := TRUE; EXIT; END_IF
END_FOR
IF NOT bFound THEN    // add if unknown
  _nPh := _nPh + 1;
  _pPh                [_nPh] := pPh;
  _nPhToPc_Mapping    [_nPh] := pMapDef^.nPc;
  _nPhToPcCh_Mapping  [_nPh] := pMapDef^.nPcCh;
  _nPhToWorker_Mapping[_nPh] := pMapDef^.nPg;
  _nPhToPgAbsoluteIdx [_nPh] := pMapDef^.nPgAbs;
ELSE
  LogWarning(F_Concat3('FB_PH=', pPh^.sName, ', already registered, ignore'));
END_IF

RegisterHw := TRUE;
END_METHOD

(*
  Container will be released (maybe destroyed) from this tracker and not available anymore after this call.
*)
METHOD remove
VAR_INPUT
	(*container at triggered event position*)
	iCT	: I_CT;
END_VAR
IF NOT bInit THEN RETURN; END_IF

// not implemented yet
END_METHOD

METHOD PROTECTED setLogLevels
VAR_INPUT
  lvl : E_LogSeverity;
END_VAR
VAR
  i : UDINT;
END_VAR
// set logging levels
fbPrintPosition.LogLevel     := lvl;
fbWorkerCamera.LogLevel      := lvl;
fbWorkerDeformation.LogLevel := lvl;
FOR i:=1 TO GVL_Maxliner.nC_MaxWorkerPrintPerPm DO
  fbWorkerPrint[i].LogLevel := lvl;
END_FOR
END_METHOD

(*
  Init/Setup print hw & link to mapped handlers.
  NOTE: override this method if it does not match the default mapping.
*)
METHOD PRIVATE SetupHw
VAR
  i : UDINT;
  sPhFdlCfg_ImgMap : ST_PH_FileDownloadCfg;
  aName : T_MaxString;
  nOldPg : UDINT;
  nPg, nPc : UDINT;
  nRelativeCtr : UDINT;
END_VAR
// check parameters
IF _iPrintGlobal.iHardwarePool = 0 THEN LogError('SetupHw: invalid hw pool reference, do not setup'); RETURN; END_IF

IF _pModuleSetup = 0 THEN LogError('Module setup not given, ignore SetupHw'); END_IF

// PC -------------------------------------------
FOR i := 1 TO _nPc DO
  // check settings
  IF _pPc[i] = 0 THEN LogError(F_Concat4('SetupHw: invalid pc mapping','_pPc[',TO_STRING(i),']=0'));
    CONTINUE;
	END_IF
  
  // build ads name
  IF nOldPg <> _nPcToPgAbsoluteIdx[i] THEN nRelativeCtr := 1; nOldPg := _nPcToPgAbsoluteIdx[i]; END_IF  // create cb counter relative to pg
  aName := F_Concat4('Controller Board', TO_STRING(_nPcToPgAbsoluteIdx[i]), '.', TO_STRING(nRelativeCtr));
  nRelativeCtr := nRelativeCtr + 1;

  // init
  _pPc[i]^.Init(    aName                 := aName
                  , sAmsNetIdLocalHost    := _pModuleSetup^.pSetupPrint^.aAmsNetId_Localhost
                  , sAmsNetIdIo           := _pModuleSetup^.pSetupPrint^.aAmsNetId_Io
                  , nEcatSlaveAddr        := TO_UINT(_pModuleSetup^.pSetupPrint^.nEcatAddr_Pc_Base + (i-1))
                  , nBlockId              := TO_INT(ePr_BLK_PC)
                  , pOd                   := _pModuleSetup^.pSetupPrint^.pOd
                  , tWaveDownload         := T#10S
                  , bHeaterEnableExist    := TRUE
                  , bPrintEnableExist     := TRUE
                  , sFilePath             := _pModuleSetup^.pSetupPrint^.aCfgPath
                  , ePcType               := E_PcTypes.Pc_RicohGen
                  );
  // register to worker
  fbWorkerPrint[_nPcToWorker_Mapping[i]].registerPc(iNewPC:=_pPc[i]^);
  
  // register to hw pool
  _iPrintGlobal.iHardwarePool.registerPc(pNewPc:=_pPc[i]);
   
END_FOR

// PH -------------------------------------------
nOldPg := 1; nRelativeCtr := 1;
FOR i := 1 TO _nPh DO
  nPc := _nPhToPc_Mapping[i];
  nPg := _nPcToPgAbsoluteIdx[nPc];
  // check config
  IF _pPh[i] = 0 OR _pPc[nPc] = 0 THEN LogError(F_Concat4('SetupHw: invalid ph mapping','_pPh[',TO_STRING(i),']=0'));
    CONTINUE;
	END_IF
  
  // build ads name
  IF nOldPg <> nPg THEN nRelativeCtr := 1; nOldPg := nPg; END_IF  // create cb counter relative to pg
  aName := F_Concat4('Printhead', TO_STRING(nPg), '.', TO_STRING(nRelativeCtr));
  nRelativeCtr := nRelativeCtr + 1;
  
  _pPh[i]^.init(    aName                 := aName
                  , sPhDef                := _pModuleSetup^.pSetupPrint^.sPHType
                  , tTempMonitor          := T#45S
                  , iChannel              := _nPhToPcCh_Mapping[i]
                  , bPositionX_Exist      := TRUE
                  , aPositionX_Unit       := 'um'
                  , lPositionX_Min        := 0
                  , lPositionX_Max        := 1_000_000
                  , bPositionY_Exist      := FALSE
                  , aPositionY_Unit       := 'pixel'
                  , lPositionY_Min        := 0
                  , lPositionY_Max        := 100_000 
                  , bShiftPositionX_Exist := FALSE      
                  , aShiftPositionX_Unit  := 'um'
                  , lShiftPositionX_Min   := 0      
                  , lShiftPositionX_Max   := 1000      
                  , bShiftPositionY_Exist := FALSE
                  , aShiftPositionY_Unit  := 'pixel'
                  , lShiftPositionY_Min   := 0
                  , lShiftPositionY_Max   := 100_000       
                  , bVoltageScale_Exist   := TRUE  
                  , aVoltageScale_Unit    := '%'
                  , fVoltageScale_Min     := 90.0  
                  , fVoltageScale_Max     := 110.0 
                  );

  _pPh[i]^.initTempMonitor(fPhTempDeviation := _pModuleSetup^.pSetupPrint^.fPhTempDeviation, tTempMonitor:=T#45S);   // overwrite default temperatur deviation
  
  // edit default file download config for ImageMap file --> disable file downloader
  _pPh[i]^.getFileDownloadConfig(E_PhFileSelection.eImageMap, stConfig=>sPhFdlCfg_ImgMap);
  sPhFdlCfg_ImgMap.bEnable := FALSE;
  _pPh[i]^.setFileDownloadConfig(eDownloader:=E_PhFileSelection.eImageMap, stConfig:=sPhFdlCfg_ImgMap);

  _pPh[i]^.LogLevel := E_LogSeverity.Info;
  
  // link ph <-> pc if not done externally
  _pPc[_nPhToPc_Mapping[i]]^.registerPH(iPH :=_pPh[i]^, nCh := TO_UINT(_nPhToPcCh_Mapping[i]));
  
  // register to worker
  fbWorkerPrint[_nPhToWorker_Mapping[i]].registerPh(iPH:=_pPh[i]^);
  
  // register to hw pool
  _iPrintGlobal.iHardwarePool.registerPh(pNewPh:=_pPh[i]);

END_FOR
END_METHOD

METHOD PRIVATE SimUpdate
VAR_INPUT
END_VAR

VAR_INST
  rfTrig_SimEnable : RF_TRIG;
END_VAR
rfTrig_SimEnable(CLK := fbSim.bSimEnable);
IF    rfTrig_SimEnable.RT THEN
  fbPrintPosition.bSimEnable := TRUE;

ELSIF rfTrig_SimEnable.FT THEN
  // ev. disable
  fbPrintPosition.bSimEnable := FALSE;
  
ELSIF fbSim.bSimEnable THEN
  // enabled
  ;
ELSE
  ; // disabled
END_IF
END_METHOD

(*
  Container triggered at position - callback.
*)
METHOD trigger : BOOL
VAR_INPUT
	sEvPos	: ST_PositionEventData;
END_VAR
IF NOT bInit THEN RETURN; END_IF
IF sEvPos.iCT = 0 THEN RETURN; END_IF


// buffer new ct
_bNewCT := TRUE;
_iNewCT := sEvPos.iCT;

LogLvl(Lvl:=E_LogSeverity.Debug, Msg:=F_Concat3(
  F_Concat2(_pModuleSetup^.aName, ' NewCT PosEv:'),
  F_Concat2(' at (Main)TrackPos:', TO_STRING(sEvPos.nTrigPos)),
  F_Concat2(' with CT:', sEvPos.iCT.print(0))
));
END_METHOD

END_FUNCTION_BLOCK

// ---- POUs/Print/Maxliner/FB_PrintModule_Maxliner_View.TcPOU
FUNCTION_BLOCK FB_PrintModule_Maxliner_View
VAR
  // helper
  bInit               : BOOL;
  
  // config
  _pModule            : POINTER TO FB_PrintModule_Maxliner;
  _pPositioning       : POINTER TO FB_PrintPositionDmax;
  
  fbCTTrackerView     : FB_CTTrackerView;
  
  // view selections
  nSelWorkerPrint     : UDINT := 1;
  bShowFineAlignement : BOOL;
  // hardware view
  bShowPhDetail       : BOOL;
  nSelPhDetail        : UDINT := 1;
  bShowPcDetail       : BOOL;
  nSelPcDetail        : UDINT := 1;
  
  // motion and position view
  bShowPositionDetail : BOOL;
  bMovingInd          : BOOL;
  fSpeed              : LREAL;
  fbBlink_Moving      : FB_BLINK;
  
  // debug view
  bShowDebugAndSim    : BOOL;
  
  fbBlink_Printing    : FB_BLINK;
  bBlinkPrint         : BOOL;
  bPrintInd           : ARRAY[1..GVL_Maxliner.nC_MaxWorkerPrintPerPm] OF BOOL;
  fMaxPos             : LREAL;
  t                   : TIME;
  zPos_PM             : UDINT;
  i                   : UDINT;
END_VAR

VAR CONSTANT
  nC_MAX_WORKER_VIEWS : UINT := 10;
END_VAR

IF NOT checkConfig() THEN RETURN; END_IF    // check config

// -- show moving -----------------------
fSpeed := _pPositioning^.getSpeed();
IF LrealIsNaN(x:=fSpeed) THEN
  fSpeed := 0;
END_IF
t := LREAL_TO_TIME(1000-fSpeed*900);
fbBlink_Moving(bI_Enable:=SEL(fSpeed > 0, FALSE, TRUE), tI_Time:=t, bO_Out=>bMovingInd);

t := T#400MS;
fbBlink_Moving(bI_Enable:=TRUE, tI_Time:=t, bO_Out=>bBlinkPrint);
FOR i:=1 TO GVL_Maxliner.nC_MaxWorkerPrintPerPm DO
  bPrintInd[i] := _pModule^.fbWorkerPrint[i].bPrinting AND bBlinkPrint;
  fMaxPos      := MAX(_pModule^.fbWorkerPrint[i].fPosition, fMaxPos);
END_FOR


// -- show pm module position
zPos_PM := SEL(_pModule^._pModuleMachineState^.bUnitInPrintPosition, 0, 40);

// -- show pg in p,
nSelWorkerPrint := LIMIT(1, nSelWorkerPrint, GVL_Maxliner.nC_MaxWorkerPrintPerPm);

// -- show ph detail
nSelPhDetail := LIMIT(1, nSelPhDetail, _pModule^._nPh);
nSelPcDetail := LIMIT(1, nSelPcDetail, _pModule^._nPc);

// -- CTTracker overview view
fbCTTrackerView.fX_m           := fMaxPos + 0.1;
fbCTTrackerView.fY_m           := 1;
fbCTTrackerView.nX_px          := 300;
fbCTTrackerView.nY_px          := 100;
fbCTTrackerView.fPxToMRatio    := fbCTTrackerView.nX_px / fbCTTrackerView.fX_m;
fbCTTrackerView.iPrintPosition :=_pPositioning^;
fbCTTrackerView();

METHOD checkConfig : BOOL
VAR_INPUT
END_VAR
VAR_INST
  _fX_m, _fY_m   : LREAL;
  _nX_px, _nY_px : DINT; 
END_VAR
VAR
  bOK : BOOL;
END_VAR
IF NOT bInit THEN RETURN; END_IF

checkConfig := TRUE;
END_METHOD

METHOD init : BOOL
VAR_INPUT
  pModule : POINTER TO FB_PrintModule_WEU;
  pPositioning : POINTER TO FB_PrintPositionDmax;
END_VAR
IF pPositioning = 0 OR pModule = 0 THEN RETURN; END_IF

_pModule      := pModule;
_pPositioning := pPositioning;

// cttracker overview
fbCTTrackerView.init(pCTTracker:=ADR(_pModule^.fbCTTracker));

bInit := TRUE;
END_METHOD

END_FUNCTION_BLOCK

// ---- POUs/Print/WEU/FB_PrintModule_WEU.TcPOU
FUNCTION_BLOCK FB_PrintModule_WEU EXTENDS FB_PrintModule_Base
VAR_INPUT
  fPUPlate1_Temperature : LREAL;  // PU Plate1 temperature
  fPUPlate2_Temperature : LREAL;  // PU Plate2 temperature
END_VAR
VAR
  (* Module specific sub-modules - WEU module contains a 
    - print position (encoder input to print domain translation)
    - Mark sensor with a mark detection module which provices a camera trigger and start position detection
    - Mark definition (used by the detection and camera)
  *)
  fbPrintPosition    : FB_PrintPositionDmax;   // a position per pm (external encoder wheel)
  fbMarkCameraWeu    : FB_MarkCamera_WEU;      // Mark detection camera
  
  // sync CT trigger with Camera detection
  _bNewCT             : BOOL;   // a new ct is received to be treated
  _iNewCT             : I_CT;   // new ct to be treated
  _bNewStartPosX0     : BOOL;   // a new startpos detected by cam
  _nNewStartPosX0     : DINT;   // new startpos X0 deteced by cam
  
  fbEncoderResoDetect : FB_EffectiveEncoderResolutionDetection;     // Effective encoder resolution detection
  fbFineAlignement    : FB_FineAlignement;     // additional grid corrections, PU Deformation/correction (4p, banana, ...)

  // messages specific
  fbMsgWeu            : ARRAY[1..nC_NumMsgWeu] OF FB_MESSAGE;  (*Messages*)
  
  // view
  fbView              : FB_PrintModule_WEU_View;    // additional controls for print module visus
END_VAR
VAR CONSTANT
  nC_NumMsgWeu        : UDINT := 6;           // number of internal messages
END_VAR

IF NOT bInit THEN RETURN; END_IF

// position
fbPrintPosition.fEnoderResolution := _pModuleMachineState^.fEncoderResolution;    // encoder resolution from machine
fbPrintPosition();

// -------------------------
// StartTrigger evaluation -> apply new CT to Tracking (created from CTM externally)
// Synchronize CT (EvPos) received from CTManger (Main) to the local StartTrigger detection and positioning
// -- reset triggers if not active
IF NOT bReadyForPrinting THEN
  _bNewCT := 0; _bNewStartPosX0 := 0;
END_IF
// -- new StartTrigger (X0)
IF bReadyForPrinting AND _iStartPos.bStartTrig AND _iStartPos.bValid THEN
  // buffer/save new start trigger
  _bNewStartPosX0 := TRUE;
  _nNewStartPosX0 := _iStartPos.nStartPositionX0;      // save detected start position for next CT to be applied to this module¨
  
  LogLvl(Lvl:=E_LogSeverity.Debug, Msg:=F_Concat3(
    F_Concat2(_pModuleSetup^.aName, ' New StartTrigger detected:'),
    F_Concat2(' at position X0:', TO_STRING(_nNewStartPosX0)),
    F_Concat2(' PM is now at: ', TO_STRING(fbPrintPosition.getPosition())),
  ));
  
  IF _bNewCT THEN   // we have an attached CT
      LogLvl(Lvl:=E_LogSeverity.Debug, Msg:=F_Concat3(
      F_Concat2(_pModuleSetup^.aName, ' Track NewCT:'),
      F_Concat2(' internal (print)Pos X0:', TO_STRING(_nNewStartPosX0)),
      F_Concat2(' with CT:', _iNewCT.print(0))
    ));
    
    _iNewCT.nPosPrint_X0 := _nNewStartPosX0;                        // set print pos to new dected in this module position domain
    fbCTTracker.RegisterCT(iCT:=_iNewCT, nX0:=_nNewStartPosX0);     // register ct for tracking in modules position and tracking system
  ELSE
    // spurious trigger (CTs not yet arrived at PMx, but receive some StartTriggers
    LogLvl(Lvl:=E_LogSeverity.Debug, Msg:=F_Concat3('StartTrigger at Pos X0:', TO_STRING(_nNewStartPosX0), ' but no CT received'));
	END_IF
  
  // reset internals (saved triggers)
  _bNewCT := FALSE; _iNewCT := 0; 
  _bNewStartPosX0 := FALSE;
END_IF

// Camera (is per module)
fbMarkCameraWeu(
  bReadyForPrinting   := bReadyForPrinting,
  nCurrentPosition    := _iPrintPosition.getPosition(),
  fCurrentSpeed       :=_iPrintPosition.getSpeed(),
  bPrintMarkExist     :=_pModuleMachineState^.bPrintMarkExist,
  bPrintDirReverse    :=_pModuleMachineState^.bPrintDirection,
  nUsePerRepeatInLine :=SEL(_pModuleMachineState^.nUsePerRepeatInLine=0, _pModuleMachineState^.nUsePerRepeatInLine, 1),
  fMarkSizeDefault    :=_pModuleMachineState^.fMarkBaseSize,
  fMarkDistRepeatToStartMark := _pModuleMachineState^.fMarkDistToStartMark,
  fMarkDistFromCenter := _pModuleMachineState^.fMarkToPrintdataCenterY
);

// Effective Encoder detection - Neutral fibre calculation with additional mark sensors
fbEncoderResoDetect(
  //bIKp_MarkTrigger01:=,
  //tIKp_TimeStampPos01:=,
  //tIKn_TimeStampNeg01:=,
  //bIKp_MarkTrigger02:=,
  //tIKp_TimeStampPos02:=,
  //tIKn_TimeStampNeg02:=,
  nPulse:=TO_DINT(fbPrintPosition.IlEncoderPulse),
  fCurrentResolution:=_pModuleMachineState^.fEncoderResolution,
  fEncoderPulseDistMin:=_pModuleMachineState^.fEncoderDetectPulseMin,
  fEncoderPulseDistMax:=_pModuleMachineState^.fEncoderDetectPulseMax,
  nDisInPulseFilterSz:=_pModuleMachineState^.nEncoderDetectFilterSz,
  fMinMarkLength:=(0.5 - 0.1) * _pModuleMachineState^.fMarkBaseSize * 1_000_000,  // 0.5*a (0*a from triangle)
  fMaxMarkLength:=(  3 + 0.1) * _pModuleMachineState^.fMarkBaseSize * 1_000_000,  //   2*a (1*a from triangle) 
  // --> the following would only work when teached
  //fMinMarkLength:=fbMarkCameraWeu.pFbMarkDefinition^.fMinMarkLength - fbMarkCameraWeu.pFbMarkDefinition^.fMarkLengthMargin * 1_000_000,
  //fMaxMarkLength:=fbMarkCameraWeu.pFbMarkDefinition^.fMaxMarkLength + fbMarkCameraWeu.pFbMarkDefinition^.fMarkLengthMargin * 1_000_000,
  //bUpdate=>,
  fDisInPulse=>_pModuleMachineFeedback^.fEncoderStepsMeasured
);

(*PU corrections*)
IF GVL_Deformation.bC_UsePUDeformation THEN
  fbFineAlignement.fT_PL1 := fPUPlate1_Temperature;
  fbFineAlignement.fT_PL2 := fPUPlate2_Temperature;
  fbFineAlignement();
END_IF

fbView();

// call module base
SUPER^();

// messages print module
fbMsgWeu[ 1](bI_Status := bTestMsg OR fbMarkCameraWeu.bMissingMarks);
fbMsgWeu[ 2](bI_Status := bTestMsg OR _pModuleMachineState^.bDriftControlMissMarks);
fbMsgWeu[ 3](bI_Status := bTestMsg OR fbMarkCameraWeu.bMarkDetectionErrors);
fbMsgWeu[ 4](bI_Status := bTestMsg OR fbMarkCameraWeu.bTeachError);
fbMsgWeu[ 5](bI_Status := bTestMsg OR fbMarkCameraWeu.bImageLengthInvalid);
fbMsgWeu[ 6](bI_Status := bTestMsg OR _bGridLimited);

IF fb_MsgQueue.bO_ReceiptMessage THEN
  fbMarkCameraWeu.ackErrors();
  _bGridLimited := FALSE;
END_IF

// simulation
SimUpdate();

PROPERTY bForceNoCorrectionButYShiftMode : BOOL
SET
FOR nCtr := 1 TO GVL_WEU.nC_MaxWorkerPrintPerPm DO
  fbWorkerPrint[nCtr].bForceNoCorrectionButShiftMode := bForceNoCorrectionButYShiftMode;
END_FOR
END_SET
END_PROPERTY

METHOD Init : BOOL
VAR_INPUT
  pModulesSetup         : POINTER TO ST_CassetteSetup;          // Module Setup Settings
  pAdsSa                : POINTER TO FB_ADS_DVTSHEETALIGNMENT;  // ADS sheet alignement
  pAdsCam               : POINTER TO FB_ADS_CAMERA;             // ADS camera
  pAdsParent            : POINTER TO FB_ADS_Config;             // Parent ADS config reference (Parent ADS block and module ref)

  // config print
  fCycleTime            : LREAL;                // task cycle time in [s]
  fPrintUnitWidth       : LREAL;                // PrintUnit width mechanical [m]
  // references
  iModule               : I_Module;             // system status interface (for sleep, estop, ...), may shadow states from machine inputs
  iPrintGlobal          : I_PrintGlobal;        // interface for module to master (main) communication
  pMachineInputs        : POINTER TO ST_ModuleMachineInterface_IN;
  pMachineOutputs       : POINTER TO ST_ModuleMachineInterface_OUT;
END_VAR
VAR
  nCtr : UDINT;
END_VAR
// Parameter checks
IF pModulesSetup = 0 OR pAdsSa = 0 OR pAdsCam = 0 OR 
    pMachineInputs = 0 OR pMachineOutputs = 0 THEN
    // set here from local fb instances: OR iModuleMaster = 0 OR iPosition = 0 OR iStartPos = 0 THEN
  LogError('init(): Invalid parameter');
  RETURN;
END_IF

// position
fbPrintPosition.Init(fPrintResolution:=pModulesSetup^.pSetupPrint^.nPrintResolution, fSubPxResolution:=pModulesSetup^.pSetupPrint^.nSubPixelResolution, fTaskCycleTime:=fCycleTime);
_iPrintPosition := fbPrintPosition;  // select reference position

// -- Mark camera
fbMarkCameraWeu.InitMarkCamera(
  fPrintUnitResolution:=_iPrintPosition.fPrintResolution, 
  fPrintUnitSubPx:=_iPrintPosition.fSubPxResolution
);
fbMarkCameraWeu.sVisuName := 'VISU_MarkCamera_WEU';
fbWorkerCamera.RegisterCamera(fbMarkCameraWeu);

// -- Sheet/Camera trigger & mark detection
_iStartPos := fbMarkCameraWeu.fbMarkDetection;  // select start position detection

SUPER^.Init(
  pModulesSetup     := pModulesSetup,
  pAdsSa            := pAdsSa,
  pAdsCam           := pAdsCam,
  pAdsParent        := pAdsParent,
  // config print
  fCycleTime        := fCycleTime,
  fPrintUnitWidth   := fPrintUnitWidth,
  // references     
  iPrintGlobal      := iPrintGlobal,     // internal subm
  iModule           := iModule, 
  pMachineInputs    := pMachineInputs,
  pMachineOutputs   := pMachineOutputs
);

// Effective Encoder Resolution detection (NeutralFibre correction)
fbEncoderResoDetect.Init();

// additional grid point corrections
fbFineAlignement.init(pAdsCam := pAdsCam, fPxReso := _iPrintPosition.fPrintResolution, fPuWidth := fPrintUnitWidth);
// - register them to workers
FOR nCtr := 1 TO GVL_WEU.nC_MaxWorkerPrintPerPm DO
  fbWorkerPrint[nCtr].RegisterGridCorrection(iGridCorrection:=fbFineAlignement);
END_FOR 

fbView.init(pModule:=THIS, pPositioning:=ADR(fbPrintPosition));
setLogLevels(lvl:=E_LogSeverity.Info);

FOR nCtr := 1 TO nC_NumMsgWeu DO
  fbMsgWeu[nCtr].pI_MsgConfig       := ADR(sL_MsgConfig);
  fbMsgWeu[nCtr].iI_MsgLocation     := 1;
END_FOR;
fbMsgWeu[ 1].iI_MsgNumber      := eCPr_PrintMarkError_Generic;        // mark detection error
fbMsgWeu[ 2].iI_MsgNumber      := eCMa_DRIFT_CONTR_ERROR;             // drift controller error
fbMsgWeu[ 3].iI_MsgNumber      := eCPr_SHEET_MARK_DETECTION;          // mark error missing/faulty
fbMsgWeu[ 4].iI_MsgNumber      := eC_STAG_CAM_TEACH_ERROR;            // teach error
fbMsgWeu[ 5].iI_MsgNumber      := eC_STAG_IMAGELENGTH_NOT_SUPPORTED;  // image length not supported (out of supported range)
fbMsgWeu[ 6].iI_MsgNumber      := eC_STAG_DEFORMATION_LIMITED;        // deformation calculated was limited to min/max before sending

Init := bInit;   // set in the SUPER class
END_METHOD

PROPERTY pMsgConfig : POINTER TO ST_MSG_CONFIG
GET
pMsgConfig := ADR(sL_MsgConfig);
END_GET
END_PROPERTY

METHOD PROTECTED setLogLevels
VAR_INPUT
  lvl : E_LogSeverity;
END_VAR
// - fb itself
LogLevel := lvl;
// - base
SUPER^.setLogLevels(lvl:=lvl);
// - weu
fbPrintPosition.LogLevel := lvl;
fbMarkCameraWeu.LogLevel := lvl;
END_METHOD

METHOD PRIVATE SimUpdate
VAR_INPUT
END_VAR
VAR_INST
  rfTrig_SimEnable : RF_TRIG;
  
  //parameter backup
  fCamMark_ToPrint, fCamMark_toDetect : LREAL;
  fCamNo_ToPrint, fCamNo_toDetect : LREAL;
END_VAR
rfTrig_SimEnable(CLK:=fbSim.bSimEnable);
IF    rfTrig_SimEnable.RT THEN
  // ev. enable
  //fbWorkerCamera.bWorkerEnable := TRUE;
  //fbWorkerDeformation.bWorkerEnable := TRUE;
  //fbWorkerPrint[1].bWorkerEnable := TRUE;
  //fbWorkerPrint[2].bWorkerEnable := TRUE;
  
  fbPrintPosition.bSimEnable  := TRUE;
  fbMarkCameraWeu.bSimulate := TRUE;

  // set some working config values
  // -backup original
  fCamMark_ToPrint  := fbMarkCameraWeu.fCameraToPrintOffset;
  fCamMark_toDetect := fbMarkCameraWeu.fDetectToCameraOffset;
  // -set sim val
  fbMarkCameraWeu.fCameraToPrintOffset := 0.4;
  fbMarkCameraWeu.fDetectToCameraOffset := 0.01;
  
  
ELSIF rfTrig_SimEnable.FT THEN
  // ev. disable
  fbPrintPosition.bSimEnable  := FALSE;
  fbMarkCameraWeu.bSimulate := FALSE;

  fbMarkCameraWeu.fCameraToPrintOffset := fCamMark_ToPrint;
  fbMarkCameraWeu.fDetectToCameraOffset := fCamMark_toDetect;
  
ELSIF fbSim.bSimEnable THEN
  // enabled
  ;
ELSE
  ; // disabled
END_IF
END_METHOD

(*
  Container triggered at position - callback.
*)
METHOD trigger : BOOL
VAR_INPUT
	sEvPos	: ST_PositionEventData;
END_VAR
IF NOT bInit THEN RETURN; END_IF
IF sEvPos.iCT = 0 THEN RETURN; END_IF


// buffer new ct
_bNewCT := TRUE;
_iNewCT := sEvPos.iCT;

LogLvl(Lvl:=E_LogSeverity.Debug, Msg:=F_Concat3(
  F_Concat2(_pModuleSetup^.aName, ' NewCT PosEv:'),
  F_Concat2(' at (Main)TrackPos:', TO_STRING(sEvPos.nTrigPos)),
  F_Concat2(' with CT:', sEvPos.iCT.print(0))
));
END_METHOD

END_FUNCTION_BLOCK

// ---- POUs/Print/Module/FB_PrintModule_Base.TcPOU
(*
  A DVT PrintModule (DEU, DSU, WEU).
*)
FUNCTION_BLOCK FB_PrintModule_Base EXTENDS T_NamedBase IMPLEMENTS I_Sim, I_PositionEvent
VAR_INPUT
  // encoder input --> directly mapped into FB_PrintPosition 
  // machine state by pointer in init()
  // external start pos interface by pointer in init()
  fPrintOffsetX           : LREAL;   // [m] external configurative offsets to PM (PU)
  fPrintOffsetY           : LREAL;   // [m] external configurative offsets to PM (PU)
END_VAR

VAR
  //config

  // - references
  _pModuleSetup           : POINTER TO ST_CassetteSetup;
  _iPrintGlobal           : I_PrintGlobal;        // master module (setting, position, global stuff, ...)
  _iPrintPosition         : I_PrintPosition;      // module's position
  _iStartPos              : I_StartPosDetect;     // module's start position detect
  _iModule                : I_Module;             // module's system status
  _pModuleMachineState    : POINTER TO ST_ModuleMachineInterface_IN;   // machine interface-print states
  _pModuleMachineFeedback : POINTER TO ST_ModuleMachineInterface_OUT;  // machine interface-print feedback
    
  // status
  bInit                   : BOOL;   // initialized
  bSelectedForPrint       : BOOL;   // selected for printing
  bReadyForPrinting       : BOOL;   // Module ready for printing
  bHardwareHold           : BOOL;   // hw hold
  _bGridLimited           : BOOL;   // calculated grid was limited before sending
  
  // instances
  fbCTTracker             : FB_CTTracker;
  fbParamMediator         : FB_DefGridParamMediator;
  fbWorkerCamera          : FB_WorkerDefGrid_Camera;
  fbWorkerDeformation     : FB_WorkerDefGrid_Deformation;
  fbWorkerPrint           : ARRAY[1..GVL_WEU.nC_MaxWorkerPrintPerPm] OF FB_WorkerDefGrid_Print_WEU;
  
  _pAdsSa                 : POINTER TO FB_ADS_DVTSHEETALIGNMENT; // sheet alignement ads
  fbAdsPm                 : FB_ADS_PM;      // PM -  Print Module ADS
  fbAdsPg                 : ARRAY[1..GVL_WEU.nC_MaxWorkerPrintPerPm] OF FB_ADS_PG;  // PG - PrintGroup ADS
  
  // hw (references only for now) ------
  // - pc
  _pPc                    : ARRAY[1..GVL_WEU.nC_MaxPcPerPm] OF POINTER TO FB_PC;
  _nPc                    : UDINT;  // number of PC in module
  _nPcToWorker_Mapping    : ARRAY[1..GVL_WEU.nC_MaxPcPerPm] OF UDINT;   // Mapping of PC to worker  
  _nPcToPgAbsoluteIdx     : ARRAY[1..GVL_WEU.nC_MaxPcPerPm] OF UDINT;   // Mapping of PC to absolute PG index
  // - ph
  _pPh                    : ARRAY[1..GVL_WEU.nC_MaxPhPerPm] OF POINTER TO FB_PH;
  _nPh                    : UDINT;  // number of PH in module
  _nPhToWorker_Mapping    : ARRAY[1..GVL_WEU.nC_MaxPhPerPm] OF UDINT;  // Mapping of PH to worker
  _nPhToPc_Mapping        : ARRAY[1..GVL_WEU.nC_MaxPhPerPm] OF UDINT;  // Mapping of PH to PC
  _nPhToPcCh_Mapping      : ARRAY[1..GVL_WEU.nC_MaxPhPerPm] OF UDINT;  // Mapping of PH to PC channel
  _nPhToPgAbsoluteIdx     : ARRAY[1..GVL_WEU.nC_MaxPhPerPm] OF UDINT;  // Mapping of PH to absolute PG index
  
  // helper
  nCtr                    : UDINT;
  nYShift_PcRamCenter     : UDINT;     // y-shift for centered image in CB RAM [px]
  fSpeed, fSpeedMpMin     : LREAL;
  bSpeedReachedForPrinting : BOOL;     // Speed for printing reached
  nPos_SubPx, nPos_Px     : DINT;
  nPos_SubPx_mem          : DINT;
  fPos_um                 : LREAL;
  nTrackPosMain           : DINT;      // tracker attach position - module position relative to pos reference in main tracker [m]

  bHwSyncCmd              : BOOL;
  sCamGridSettings        : ST_CameraGridSettings;
  bOnePgActive            : BOOL;

    
  // messaging
  fb_MsgQueue             : FB_MSG_QUEUE;                 (*Message queue*)
  fb_MsgHandler           : FB_MSG_HANDLER;               (*Message handler*)
  sL_MsgConfig            : ST_MSG_CONFIG;                (*Message config*)
  //fbMsg                   : ARRAY [1..nC_NumMsg] OF FB_MESSAGE;  (*Messages*)
  
  // simulation
  fbSim                   : FB_Sim;
  // test
  bTestMsg : BOOL;      // activate message test
END_VAR
VAR PERSISTENT
  _fPmDistToPrev          : LREAL;                 // [m] distance to previous PM (in main domain)
  _fPmMainTrackPos        : LREAL;                 // [m] used distance to master reference position (in main tracker)
END_VAR
VAR CONSTANT
  nC_NumMsg               : UDINT := 0;            // number of internal messages
  fC_HeadOffsetPlate      : LREAL := 0.000_2;      // Head offset to base plate [m] (mechanical)
  fC_MinimalProductionSpeed_in_MpMin: LREAL := 5.0;    // [m/min]
  fC_FormatLengthTolerance : LREAL := 100.0;       // [px] tolerance of substrate length job - machine config 
  nC_StopReadyTimeout     : TIME := T#10S;         // Synced stopping of printing, max. timeout to wait for printing end
END_VAR

IF NOT bInit THEN RETURN; END_IF

// positioning
// - get position 
nPos_SubPx := _iPrintPosition.getPosition(nPosition_px=>nPos_Px, fPosition_um=>fPos_um);
// (disabled) nPos_SubPx := nPos_SubPx_mem := SEL(bReadyForPrinting AND _iPrintPosition.bMoving, nPos_SubPx_mem, nPos_SubPx);   // security measure (jetting when not really moving or not in position
// - get speed
fSpeed := _iPrintPosition.getSpeed(fSpeedMpMin=>fSpeedMpMin);

// update distance from machine
_fPmDistToPrev := _pModuleMachineState^.fDistanceToPrevModule;

// enable, control, release signals
//   engaged -> selected and prepared for production
//   printActivated -> machine & axis position ready for printing
//   InitInPrintPosition -> module in pos to allow printing
bSelectedForPrint        := fbAdsPm.bEnable AND _pModuleMachineState^.bEngaged;
bSpeedReachedForPrinting := (fSpeedMpMin >= fC_MinimalProductionSpeed_in_MpMin);
// ready for printing (enable detection)
bReadyForPrinting        :=      bSelectedForPrint                                // selected and ready for production (from machine)
                            AND _pModuleMachineState^.bPrintActivated             // machine & axis ready for printing
                            AND _pModuleMachineState^.bUnitInPrintPosition        // module in printing position -> allowed to print
                            AND bSpeedReachedForPrinting                          // speed bigger than min speed for printing
                            AND _pModuleMachineState^.bTargetSpeedReached         // do not evaluate marks while machine ramping up  
                            AND NOT _pModuleMachineState^.bStopRequest            // do not evaluate marks while machine is stopping
                            AND NOT _pModuleMachineState^.bEStop
                            AND NOT _pModuleMachineState^.bSleep;
bHardwareHold            := NOT bSpeedReachedForPrinting OR 
                            NOT _pModuleMachineState^.bPrintActivated OR 
                            NOT _pModuleMachineState^.bUnitInPrintPosition OR 
                                _pModuleMachineState^.bFastStopRequest;
bHwSyncCmd               := checkHwSyncRequest();                                 // sync trigger generation

// pos for attach in main tracker
nTrackPosMain := F_MeterToSubPixel(fPosMeter:=_fPmMainTrackPos, fResoSubPx:=_iPrintPosition.fPrintResolution*_iPrintPosition.fSubPxResolution); 
// run tracker
fbCTTracker(nPos:=nPos_SubPx);


// call hardware
(* -- PC PrintController*)
FOR nCtr := 1 TO _nPc DO
  IF _pPc[nCtr] <> 0 THEN
    _pPc[nCtr]^.sI_SystemCmd.bSleep := _pModuleMachineState^.bSleep;  // from if to module (machine)
    _pPc[nCtr]^.sI_SystemCmd.bEStop := _pModuleMachineState^.bEStop;  // from if to module (machine)
    _pPc[nCtr]^.sI_SystemCmd.bAirNotOk := FALSE;
    _pPc[nCtr]^();
  END_IF
END_FOR

(* -- PH PrintHead*)
FOR nCtr := 1 TO _nPh DO
  IF _pPh[nCtr] <> 0 THEN
    ; // called in PC.update()->pPh[nCtr]^();
  END_IF
END_FOR


// Worker
// - Camera
fbWorkerCamera.bWorkerEnable := fbAdsPm.bEnable AND bOnePgActive;
sCamGridSettings := fbWorkerCamera.sCameraGridSettings;
// - Deformation
fbWorkerDeformation.bWorkerEnable := fbAdsPm.bEnable AND bOnePgActive AND sCamGridSettings.eDeformationType > E_DeformationType.NoDeformation;

// - Print
// - fill I_SubSystem correctly from all workers
FOR nCtr := 1 TO GVL_WEU.nC_MaxWorkerPrintPerPm DO
  fbWorkerPrint[nCtr].bWorkerEnable := fbAdsPm.bEnable AND fbWorkerPrint[nCtr]._pAdsPg^.bEnable;
  fbWorkerPrint[nCtr].bWorkerPrintEnable := _pModuleMachineState^.bPrintActivated;
  fbWorkerPrint[nCtr](
    nPrintPos             := nPos_SubPx,
    fMasterSpeed          := fSpeed,
    bHardwareSync         := bHwSyncCmd,
    bHardwareHold         := bHardwareHold,
    bFastStopRequest      := _pModuleMachineState^.bFastStopRequest,
    bPrintStopRequest     := _pModuleMachineState^.bStopRequest,
                            // Print StartPosition Distance to detected X0 of CT
    fPrintStartOffset     :=   fPrintOffsetX                                    // NOTE: dynamic corrections done in Worker (dropSpeedComp / global grid dx / other point corrections))
                             - TO_LREAL(fbAdsPm.nGeneralShiftX) / 1_000_000     // ! negative direction to match PUC UI => change requested by STAG (14.08.2024)
                             + TO_LREAL(fbAdsPg[nCtr].nPositionX) / 1_000_000,
    fPrintYOffset         := LIMIT(
                              0,
                                F_SubPixelToMeter(TO_DINT(nYShift_PcRamCenter), _iPrintPosition.fPrintResolution)              // y-offset for centered image in ph
                                + fPrintOffsetY
                                - TO_LREAL(fbAdsPm.nGeneralShiftY) / 1_000_000    // ! negative direction to match PUC UI => change requested by STAG (16.12.2024)
                                + TO_LREAL(fbAdsPg[nCtr].nPositionY) / 1_000_000
                                + _pModuleMachineState^.fLateralRegister  // lateral register from machine
                              ,2*F_SubPixelToMeter(TO_DINT(nYShift_PcRamCenter), _iPrintPosition.fPrintResolution)
                            ),
    nPhDepth              := _pModuleSetup^.pSetupPrint^.sPHType.iC_Ph_Depth,
    fPUElevation          := _pModuleMachineFeedback^.fHeadGap, // + fC_HeadOffsetPlate,
//    bError                => ,
//    nError                => ,
  );
END_FOR

// collect printWorker status
FOR nCtr := 1 TO GVL_WEU.nC_MaxWorkerPrintPerPm DO
  IF fbWorkerPrint[nCtr].bWorkerEnable THEN
    _bGridLimited := fbWorkerPrint[nCtr].bGridWasLimited OR _bGridLimited; 
	END_IF
END_FOR

// One PG (printWorker) active
bOnePgActive := FALSE;
FOR nCtr := 1 TO GVL_WEU.nC_MaxWorkerPrintPerPm DO 
  IF fbAdsPg[nCtr].bEnable THEN bOnePgActive := TRUE; END_IF 
END_FOR

  
// machine interface outputs
_pModuleMachineFeedback^.bMoving           := bSpeedReachedForPrinting;
_pModuleMachineFeedback^.fSpeed            := fSpeed;
_pModuleMachineFeedback^.fPosition         := fPos_um / 1_000_000;
_pModuleMachineFeedback^.bSpeedExeeded     := checkSpeed(fSpeed:=fSpeed, fMaxSpeed => _pModuleMachineFeedback^.fMaxSpeed);
_pModuleMachineFeedback^.bLengthMismatch   := checkFormatLength();
_pModuleMachineFeedback^.bStopReady        := checkReadyForStop(bStopRequestSync:=_pModuleMachineState^.bStopRequest);
_pModuleMachineFeedback^.fHeadGap          := _pAdsSa^.fHeadGap / 1000;  // [mm] -> [m]
_pModuleMachineFeedback^.fInkQuantity      := getInkQuantity();

// messaging
Messaging();

{attribute 'monitoring':='call'}
PROPERTY bMoving : BOOL
GET
bMoving := _iPrintPosition.bMoving;
END_GET
END_PROPERTY

{attribute 'monitoring' := 'call'}
// module is selected for production (and considered in positioning)
PROPERTY bSelectedForProduction : BOOL
GET
bSelectedForProduction := bSelectedForPrint;
END_GET
END_PROPERTY

{attribute 'monitoring' := 'call'}
(*Simulation is enabled set/get*)
PROPERTY bSimEnable : BOOL
GET
bSimEnable := fbSim.bSimEnable;
END_GET
SET
fbSim.bSimEnable := bSimEnable;
END_SET
END_PROPERTY

(* 
  Hardware sync request.
*)
PROPERTY bSyncCmd : BOOL
GET
bSyncCmd := bHwSyncCmd;
END_GET
END_PROPERTY

// check imagelength vs formatlength
// :returns: TRUE if a mismatch was detected
METHOD PRIVATE checkFormatLength : BOOL
VAR 
  nFormatTolerance : LREAL;
  bOneJobActive    : BOOL;
  i                : UDINT;
  _fImageLength    : LREAL;
END_VAR
// check config
_fImageLength := 0;
FOR i := 1 TO GVL_WEU.nC_MaxWorkerPrintPerPm DO
  IF fbWorkerPrint[i]._bEnable THEN
    _fImageLength := fbWorkerPrint[i].fImageLength;
	END_IF
END_FOR

IF _fImageLength = 0 THEN RETURN; END_IF
IF _pModuleMachineState^.fSubstrateLen = 0 THEN RETURN; END_IF
IF bSimEnable THEN RETURN; END_IF  // check ok during simulation

bOneJobActive := FALSE;
FOR i := 1 TO GVL_WEU.nC_MaxWorkerPrintPerPm DO
  bOneJobActive := bOneJobActive OR fbWorkerPrint[i].bJobActive;
END_FOR
IF NOT bOneJobActive THEN RETURN; END_IF

// compare
nFormatTolerance := fC_FormatLengthTolerance / _pModuleSetup^.pSetupPrint^.nPrintResolution * 0.0254;  // 100 [px] -> [m]
IF nFormatTolerance < ABS(_fImageLength - _pModuleMachineState^.fSubstrateLen) THEN
  checkFormatLength := TRUE;
END_IF
END_METHOD

METHOD PROTECTED checkHwSyncRequest : BOOL
VAR_INST
  rT_SyncRequest : R_TRIG;
  tSyncDelay     : TON;
END_VAR
VAR_OUTPUT
  bHwSyncReq : BOOL;
END_VAR
rT_SyncRequest(CLK:=bReadyForPrinting);
IF rT_SyncRequest.Q OR _iPrintPosition.bStarted THEN  // OR rT_JobActive.Q 
  tSyncDelay(IN:=TRUE, PT:=T#2MS);   // a Sync delay to workaround a sync sent to CB while a Start or Prepare Command
END_IF
tSyncDelay(Q=>bHwSyncReq);
IF tSyncDelay.Q THEN 
  tSyncDelay(IN:=FALSE);
END_IF


checkHwSyncRequest := bHwSyncReq;
END_METHOD

METHOD PRIVATE checkReadyForStop : BOOL
VAR_INPUT
  bStopRequestSync : BOOL;
END_VAR
VAR
  i : UDINT;
  bStopReady : BOOL;
END_VAR
VAR_INST
  tOnStoppingSupversion : TON;  // check if it takes too long for stopping print with (synced)stop-request
  rTSupervsion : R_TRIG;
END_VAR
// check print states
bStopReady := TRUE;
FOR i := 1 TO GVL_WEU.nC_MaxWorkerPrintPerPm DO                        // all worker stopped?
  bStopReady := bStopReady AND NOT fbWorkerPrint[i].bPrintActive;   // stop ready if no print is active
END_FOR

// error handling
// - 
tOnStoppingSupversion(IN:=bStopRequestSync AND NOT bStopReady, PT:=nC_StopReadyTimeout);   // supervision for synchronized stopping the print of module
rTSupervsion(CLK:=bStopRequestSync AND tOnStoppingSupversion.Q);    // 
IF rTSupervsion.Q THEN LogWarning('checkReadyForStop: stopped by timeout (stop ready not received from PM)'); END_IF


// ready if request set and all finished printing (or supervision)
checkReadyForStop := bStopRequestSync AND (bStopReady OR tOnStoppingSupversion.Q);
END_METHOD

(*
  Checks if current speed is higher than max. speed.
  :return: TRUE if speed exeeds maximum
*)
METHOD PROTECTED checkSpeed : BOOL
VAR_INPUT
  fSpeed : LREAL;       // current speed
END_VAR
VAR_OUTPUT
  fMaxSpeed : LREAL;    // modules max. printing speed
END_VAR
VAR
  f : LREAL;
  i : UDINT;
END_VAR
VAR_INST
  fbSpeedFilterMav : FB_FILTER_MAV;           // Moving average filter
  fMaxSpeedTolerence : LREAL := 1.0/60;       // Allow max. speed to exeed limit + this tolerance 
END_VAR
// disabled
IF NOT fbAdsPm.bEnable OR NOT _pModuleMachineState^.bEngaged THEN 
  checkSpeed := FALSE;
  fMaxSpeed := 0;
  RETURN;
END_IF 


// filter current speed
fbSpeedFilterMav(fI_Input := fSpeed, iI_NbInputs := 32);  (*max iI_NbInputs = 32!*)

// find slowest max. speed
f := 0;
FOR i:=1 TO GVL_WEU.nC_MaxWorkerPrintPerPm DO
  IF fbWorkerPrint[i].bWorkerEnable THEN
    IF fbWorkerPrint[i].fMaxSpeed = 0 THEN
      ; // ignored speed
    ELSIF f = 0 OR f > fbWorkerPrint[i].fMaxSpeed THEN 
      f := fbWorkerPrint[i].fMaxSpeed;
		END_IF
	END_IF
END_FOR

fMaxSpeed := f;   // return max. possible speed

// check if too fast
IF f > 0 AND fbSpeedFilterMav.fO_OutputMav > (f+fMaxSpeedTolerence) THEN 
  checkSpeed := TRUE; // speed exceeded
ELSE
  checkSpeed := FALSE;
END_IF
END_METHOD

(*
  Distance between activated StartPosition detection and Pm, if one configured (fDetectToCameraOffset + fCameraToPrintOffset)
  If no StartPos detection = 0
*)
PROPERTY fDetectToPm : LREAL
GET
fDetectToPm := fbWorkerCamera.fDetectToCamOffset + fbWorkerCamera.fCameraToPrintOffset;
END_GET
END_PROPERTY

// distance to previous print module (on master tracking pos)
PROPERTY fPmDistToPrev : LREAL
GET
fPmDistToPrev := _fPmDistToPrev;
END_GET
SET
_fPmDistToPrev := fPmDistToPrev;
END_SET
END_PROPERTY

PROPERTY fPmMainTrackPos : LREAL
GET
fPmMainTrackPos := _fPmMainTrackPos;
END_GET
SET
_fPmMainTrackPos := fPmMainTrackPos;
END_SET
END_PROPERTY

METHOD getInkQuantity : LREAL
VAR
  nWorker : UDINT;
END_VAR
FOR nWorker := 1 TO GVL_WEU.nC_MaxWorkerPrintPerPm DO
  IF fbWorkerPrint[nWorker].bWorkerEnable THEN    // from first enabled worker (PG)
    getInkQuantity := fbWorkerPrint[nWorker]._pAdsPg^.lInkQuantity;
    EXIT;
	END_IF
END_FOR
END_METHOD

METHOD Init : BOOL
VAR_INPUT
  pModulesSetup         : POINTER TO ST_CassetteSetup;          // Module Setup Settings
  pAdsSa                : POINTER TO FB_ADS_DVTSHEETALIGNMENT;  // ADS sheet alignement
  pAdsCam               : POINTER TO FB_ADS_CAMERA;             // ADS camera
  pAdsParent            : POINTER TO FB_ADS_Config;             // Parent ADS config reference (Parent ADS block and module ref)

  // config print
  fCycleTime            : LREAL;                // task cycle time in [s]
  fPrintUnitWidth       : LREAL;                // PrintUnit width mechanical [m]
  // references
  iModule               : I_Module;             // system status interface (for sleep, estop, ...), may shadow states from machine inputs
  iPrintGlobal          : I_PrintGlobal;        // interface for module to master (main) communication
  pMachineInputs        : POINTER TO ST_ModuleMachineInterface_IN;
  pMachineOutputs       : POINTER TO ST_ModuleMachineInterface_OUT;
END_VAR
VAR
  nCtr : UDINT;
  sMode : ST_SimModeDef;
END_VAR
IF  pModulesSetup = 0 OR pAdsSa = 0 OR pAdsCam = 0 OR pAdsParent = 0 OR 
    pMachineInputs = 0 OR pMachineOutputs = 0 OR
    iPrintGlobal = 0 THEN
  LogError('init(): Invalid parameter');
  RETURN;
END_IF

// save config
_pModuleSetup := pModulesSetup;
_pAdsSa := pAdsSa;
_iPrintGlobal := iPrintGlobal;
_iModule := iModule;
_pModuleMachineState := pMachineInputs;
_pModuleMachineFeedback := pMachineOutputs;
nYShift_PcRamCenter := _pModuleSetup^.pSetupPrint^.nPcYShiftCenterRam;

// init & setup hw and module linking
SetupHw();

// ADS config and mapping
InitAds(pAdsParent:=pAdsParent);

// cttracker
fbCTTracker.Init(aName:=F_Concat2('Tracker of ', pModulesSetup^.aName), aUnit:='SubPx', bAutoRemoveAfterLastEvPos:=TRUE);

// Worker
// -- parameter mediator
fbParamMediator.init(pCamWorker:=ADR(fbWorkerCamera), pDefWorker:=ADR(fbWorkerDeformation));

// -- Worker camera
fbWorkerCamera.Init(pMsgConfig:=ADR(sL_MsgConfig), fPrintResolution:=_iPrintPosition.fPrintResolution, fSubPxResolution:=_iPrintPosition.fSubPxResolution, bParallelCT:=TRUE);
fbWorkerCamera.InitWorkerCamera(pAdsIf:=pAdsCam, iDefGridParamMediator:=fbParamMediator, fFeatureGrid:=256, fPrintUnitWidth:=fPrintUnitWidth);
fbWorkerCamera.reg();
fbCTTracker.RegisterTrackPos(iPositionEvent:=fbWorkerCamera);
iPrintGlobal.registerPuStatusClient(sClient:=fbWorkerCamera);

// -- Worker deformation
fbWorkerDeformation.Init(pMsgConfig:=ADR(sL_MsgConfig), fPrintResolution:=_iPrintPosition.fPrintResolution, fSubPxResolution:=_iPrintPosition.fSubPxResolution, bParallelCT:=TRUE);
fbWorkerDeformation.InitWorkerDeformation(nPrintUnitWidth:=TO_UDINT(F_MeterToSubPixel(fPosMeter:=fPrintUnitWidth, fResoSubPx:=_iPrintPosition.fPrintResolution)), iDefGridParamMediator:=fbParamMediator);
fbWorkerDeformation.reg();
fbCTTracker.RegisterTrackPos(iPositionEvent:=fbWorkerDeformation);
iPrintGlobal.registerPuStatusClient(sClient:=fbWorkerDeformation);

// -- Worker print
FOR nCtr := 1 TO GVL_WEU.nC_MaxWorkerPrintPerPm DO
  fbWorkerPrint[nCtr].Init(
    fPrintResolution:=_iPrintPosition.fPrintResolution,
    fSubPxResolution:=_iPrintPosition.fSubPxResolution,
    pMsgConfig:=ADR(sL_MsgConfig),
    bParallelCT:=TRUE
  );
  fbWorkerPrint[nCtr].InitWorkerPrint(
    pAdsPg:=ADR(fbAdsPg[nCtr]),
    iDefGridParamMediator:=fbParamMediator,
    fLimitCorrectionX:=1000,
    fLimitCorrectionY:=nYShift_PcRamCenter-1
  );
  fbWorkerPrint[nCtr].reg();
  fbCTTracker.RegisterTrackPos(iPositionEvent:=fbWorkerPrint[nCtr]);
  iPrintGlobal.registerPuSubystem(iSubSys:=fbWorkerPrint[nCtr]);
END_FOR

(*Messaging*)
sL_MsgConfig.bI_Enable       := TRUE;
sL_MsgConfig.pI_FbMsgHandler := ADR(fb_MsgHandler);
fb_MsgHandler.pI_MsgQueue    := ADR(fb_MsgQueue);
fb_MsgQueue.pI_MsgInterface  := fbAdsPm.pMsgInterface;
fb_MsgQueue.cI_MaxElement    := TO_INT(SIZEOF(fbAdsPm.pMsgInterface^.sO_MsgBuffer)/SIZEOF(ST_ADS_MSG));

(*Messages*)
(*
FOR nCtr := 1 TO nC_NumMsg DO
  fbMsg[nCtr].pI_MsgConfig   := ADR(sL_MsgConfig);
  fbMsg[nCtr].iI_MsgLocation := 1;
END_FOR;

fbMsg[ 1].iI_MsgNumber       := ;     // mark detection error
*)
Init := bInit := TRUE;
END_METHOD

// ADS Configuration of interface 
// ADS Block Mapping of Module
METHOD PROTECTED InitAds
VAR_INPUT
  pAdsParent  : POINTER TO FB_ADS_Config;             // Parent ADS config reference (Parent ADS block and module ref)
END_VAR
// ADS Mapping --------------------------------------------
// -> to PU
pAdsParent^.register(ADR(fbAdsPm));  // PM -->PU
// -> to PM
FOR nCtr := 1 TO GVL_WEU.nC_MaxWorkerPrintPerPm DO
  pAdsParent^.iAdsParent := fbAdsPm;
  pAdsParent^.register(ADR(fbAdsPg[nCtr]));    // PG --> PM
  (*groups -> header tank group*)
  pAdsParent^.iAdsParent := _pModuleSetup^.pSetupInk^.pInkHeaderTankGroup^;
  pAdsParent^.register(ADR(fbAdsPg[nCtr]));    // PG --> HT Group
END_FOR

// -> to PG
FOR nCtr := 1 TO _nPc DO
  pAdsParent^.iAdsParent := fbAdsPg[_nPcToWorker_Mapping[nCtr]];
  pAdsParent^.register(_pPc[nCtr]^.pAdsBlock);     // PC --> PG
END_FOR;

// -> to PC
(*printhead*)
FOR nCtr := 1 TO _nPh DO
  pAdsParent^.iAdsParent := _pPc[_nPhToPc_Mapping[nCtr]]^.pAdsBlock^;
  pAdsParent^.register(_pPh[nCtr]^.pAdsBlock);    // PH --> PC
END_FOR;


// ADS Config ---------------------------------------------
(* -- PM PrintModuile*)
fbAdsPm.aName := _pModuleSetup^.aName;
fbAdsPm.config(
    bGeneralShiftX_Exist := TRUE
  , aGeneralShiftX_Unit  :=  'um'
  , nGeneralShiftX_Min   := -380_000
  , nGeneralShiftX_Max   := 1_000_000
  
  , bGeneralShiftY_Exist := TRUE
  , aGeneralShiftY_Unit  := 'um'
  , nGeneralShiftY_Min   := -8_001
  , nGeneralShiftY_Max   := 8_001
);

(* -- PG PrintGroup*)
FOR nCtr := 1 TO GVL_WEU.nC_MaxWorkerPrintPerPm DO
  fbAdsPg[nCtr].aName := F_Concat4(fbAdsPm.aName, ' - ', 'Printline ', TO_STRING(nCtr));
  fbAdsPg[nCtr].config(
       bShiftPositionX_Exist     := TRUE
     , aShiftPositionX_Unit      := 'um'
     , lShiftPositionX_Min       := 0
     , lShiftPositionX_Max       := 2_000_000
     
     , bShiftPositionY_Exist     := FALSE
     , aShiftPositionY_Unit      := 'pixel'
     , lShiftPositionY_Min       := 0
     , lShiftPositionY_Max       := 2147483647
     
     , bInkQuantity_Exist        := FALSE
     , aInkQuantity_Unit         := 'g/m^2'
     , lInkQuantity_Min          := 0
     , lInkQuantity_Max          := 100
     
     , bMaxPrintSpeed_Exist      := FALSE
     , aMaxPrintSpeed_Unit       := 'm/min'
     , lMaxPrintSpeed_Min        := 0
     , lMaxPrintSpeed_Max        := 100
  );
END_FOR;
END_METHOD

PROPERTY iPrintPosition : I_PrintPosition
GET
iPrintPosition := _iPrintPosition;
END_GET
END_PROPERTY

PROPERTY iStartPos : I_StartPosDetect
GET
iStartPos := _iStartPos;
END_GET
END_PROPERTY

METHOD PRIVATE Messaging
VAR_INPUT
END_VAR
(*Messaging*)
fb_MsgHandler();
fb_MsgQueue();

// messages print module
//fbMsg[ 1](bI_Status := bTestMsg OR );

// message ack
IF fb_MsgQueue.bO_ReceiptMessage THEN
  IF bTestMsg THEN LogInfo('Ack messages'); END_IF
END_IF
END_METHOD

PROPERTY nTrackOffset : DINT
GET
nTrackOffset := nTrackPosMain;
END_GET
END_PROPERTY

(*
  NOTE: Only needed because the Hw instances are outside of the Module.
        Please call the register HW prior initializing the Module itself!
*)
METHOD RegisterHw : BOOL
VAR_INPUT
  pPh : POINTER TO FB_PH;
  pPc : POINTER TO FB_PC;
  pMapDef : POINTER TO ST_MappingDefinition;
END_VAR
VAR
  i : UDINT;
  bFound : BOOL;
END_VAR
IF pPh = 0 OR pPc = 0 OR pMapDef = 0 THEN LogError('registerHw invalid parameter'); RETURN; END_IF
IF _nPc >= GVL_WEU.nC_MaxPcPerPm THEN LogError('register hw: too many PCs registered'); RETURN; END_IF
IF _nPh >= GVL_WEU.nC_MaxPhPerPm THEN LogError('register hw: too many PHs registered'); RETURN; END_IF

// PC 
bFound := FALSE;
FOR i:=1 TO _nPc DO   // search for existing pc
  IF _pPc[i] = pPc THEN bFound := TRUE; EXIT; END_IF
END_FOR
IF NOT bFound THEN    // add if unknown
  _nPc := _nPc + 1;
  _pPc[_nPc] := pPc;
  _nPcToWorker_Mapping[_nPc] := pMapDef^.nPg;  // save mapping
  _nPcToPgAbsoluteIdx[_nPc] := pMapDef^.nPgAbs;  // save PCs mapping to PG absolute
ELSE
  ; // ignore new pc
END_IF

// PH
bFound := FALSE;
FOR i:=1 TO _nPh DO   // search for existing ph
  IF _pPh[i] = pPh THEN bFound := TRUE; EXIT; END_IF
END_FOR
IF NOT bFound THEN    // add if unknown
  _nPh := _nPh + 1;
  _pPh[_nPh] := pPh;
  _nPhToPc_Mapping[_nPh] := pMapDef^.nPc;
  _nPhToPcCh_Mapping[_nPh] := pMapDef^.nPcCh;
  _nPhToWorker_Mapping[_nPh] := pMapDef^.nPg;
  _nPhToPgAbsoluteIdx[_nPh] := pMapDef^.nPgAbs;
ELSE
  LogWarning(F_Concat3('FB_PH=', pPh^.sName, ', already registered, ignore'));
END_IF

RegisterHw := TRUE;
END_METHOD

(*
  Container will be released (maybe destroyed) from this tracker and not available anymore after this call.
*)
METHOD remove
VAR_INPUT
	(*container at triggered event position*)
	iCT	: I_CT;
END_VAR
IF NOT bInit THEN RETURN; END_IF

// not implemented yet
END_METHOD

METHOD PROTECTED setLogLevels
VAR_INPUT
  lvl : E_LogSeverity;
END_VAR
VAR
  i : UDINT;
END_VAR
// set logging levels
fbWorkerCamera.LogLevel := lvl;
fbWorkerDeformation.LogLevel := lvl;
FOR i:=1 TO GVL_WEU.nC_MaxWorkerPrintPerPm DO
  fbWorkerPrint[i].LogLevel := lvl;
END_FOR
END_METHOD

(*
  Init/Setup print hw & link to mapped handlers.
  NOTE: override this method if it does not match the default mapping.
*)
METHOD PRIVATE SetupHw
VAR
  i : UDINT;
  sPhFdlCfg_ImgMap : ST_PH_FileDownloadCfg;
  aName : T_MaxString;
  nOldPg : UDINT;
  nPg, nPc : UDINT;
  nRelativeCtr : UDINT;
END_VAR
// check parameters
IF _iPrintGlobal.iHardwarePool = 0 THEN LogError('SetupHw: invalid hw pool reference, do not setup'); RETURN; END_IF

IF _pModuleSetup = 0 THEN LogError('Module setup not given, ignore SetupHw'); END_IF

// PC -------------------------------------------
FOR i := 1 TO _nPc DO
  // check settings
  IF _pPc[i] = 0 THEN LogError(F_Concat4('SetupHw: invalid pc mapping','_pPc[',TO_STRING(i),']=0'));
    CONTINUE;
	END_IF
  
  // build ads name
  IF nOldPg <> _nPcToPgAbsoluteIdx[i] THEN nRelativeCtr := 1; nOldPg := _nPcToPgAbsoluteIdx[i]; END_IF  // create cb counter relative to pg
  aName := F_Concat4('Controller Board', TO_STRING(_nPcToPgAbsoluteIdx[i]), '.', TO_STRING(nRelativeCtr));
  nRelativeCtr := nRelativeCtr + 1;

  // init
  _pPc[i]^.Init(    aName                 := aName
                  , sAmsNetIdLocalHost    := _pModuleSetup^.pSetupPrint^.aAmsNetId_Localhost
                  , sAmsNetIdIo           := _pModuleSetup^.pSetupPrint^.aAmsNetId_Io
                  , nEcatSlaveAddr        := TO_UINT(_pModuleSetup^.pSetupPrint^.nEcatAddr_Pc_Base + (i-1))
                  , nBlockId              := TO_INT(ePr_BLK_PC)
                  , pOd                   := _pModuleSetup^.pSetupPrint^.pOd
                  , tWaveDownload         := T#10S
                  , bHeaterEnableExist    := TRUE
                  , bPrintEnableExist     := TRUE
                  , sFilePath             := _pModuleSetup^.pSetupPrint^.aCfgPath
                  , ePcType               := E_PcTypes.Pc_RicohGen
                  );
  // register to worker
  fbWorkerPrint[_nPcToWorker_Mapping[i]].registerPc(iNewPC:=_pPc[i]^);
  
  // register to hw pool
  _iPrintGlobal.iHardwarePool.registerPc(pNewPc:=_pPc[i]);
   
END_FOR

// PH -------------------------------------------
nOldPg := 1; nRelativeCtr := 1;
FOR i := 1 TO _nPh DO
  nPc := _nPhToPc_Mapping[i];
  nPg := _nPcToPgAbsoluteIdx[nPc];
  // check config
  IF _pPh[i] = 0 OR _pPc[nPc] = 0 THEN LogError(F_Concat4('SetupHw: invalid ph mapping','_pPh[',TO_STRING(i),']=0'));
    CONTINUE;
	END_IF
  
  // build ads name
  IF nOldPg <> nPg THEN nRelativeCtr := 1; nOldPg := nPg; END_IF  // create cb counter relative to pg
  aName := F_Concat4('Printhead', TO_STRING(nPg), '.', TO_STRING(nRelativeCtr));
  nRelativeCtr := nRelativeCtr + 1;
  
  _pPh[i]^.init(    aName                 := aName
                  , sPhDef                := _pModuleSetup^.pSetupPrint^.sPHType
                  , tTempMonitor          := T#45S
                  , iChannel              := _nPhToPcCh_Mapping[i]
                  , bPositionX_Exist      := TRUE
                  , aPositionX_Unit       := 'um'
                  , lPositionX_Min        := 0
                  , lPositionX_Max        := 1_000_000
                  , bPositionY_Exist      := FALSE
                  , aPositionY_Unit       := 'pixel'
                  , lPositionY_Min        := 0
                  , lPositionY_Max        := 100_000 
                  , bShiftPositionX_Exist := FALSE      
                  , aShiftPositionX_Unit  := 'um'
                  , lShiftPositionX_Min   := 0      
                  , lShiftPositionX_Max   := 1000      
                  , bShiftPositionY_Exist := FALSE
                  , aShiftPositionY_Unit  := 'pixel'
                  , lShiftPositionY_Min   := 0
                  , lShiftPositionY_Max   := 100_000       
                  , bVoltageScale_Exist   := TRUE  
                  , aVoltageScale_Unit    := '%'
                  , fVoltageScale_Min     := 90.0  
                  , fVoltageScale_Max     := 110.0 
                  );

  _pPh[i]^.initTempMonitor(fPhTempDeviation := _pModuleSetup^.pSetupPrint^.fPhTempDeviation, tTempMonitor:=T#45S);   // overwrite default temperatur deviation
  
  // edit default file download config for ImageMap file --> disable file downloader
  _pPh[i]^.getFileDownloadConfig(E_PhFileSelection.eImageMap, stConfig=>sPhFdlCfg_ImgMap);
  sPhFdlCfg_ImgMap.bEnable := FALSE;
  _pPh[i]^.setFileDownloadConfig(eDownloader:=E_PhFileSelection.eImageMap, stConfig:=sPhFdlCfg_ImgMap);

  _pPh[i]^.LogLevel := E_LogSeverity.Info;
  
  // link ph <-> pc if not done externally
  _pPc[_nPhToPc_Mapping[i]]^.registerPH(iPH :=_pPh[i]^, nCh := TO_UINT(_nPhToPcCh_Mapping[i]));
  
  // register to worker
  fbWorkerPrint[_nPhToWorker_Mapping[i]].registerPh(iPH:=_pPh[i]^);
  
  // register to hw pool
  _iPrintGlobal.iHardwarePool.registerPh(pNewPh:=_pPh[i]);

END_FOR
END_METHOD

(*
  Container triggered at position - callback.
*)
METHOD trigger : BOOL
VAR_INPUT
	sEvPos	: ST_PositionEventData;
END_VAR
IF NOT bInit THEN RETURN; END_IF

// not implemented --> see child
END_METHOD

END_FUNCTION_BLOCK

// ---- POUs/Print/WEU/FB_WorkerDefGrid_Print_WEU.TcPOU
FUNCTION_BLOCK FB_WorkerDefGrid_Print_WEU EXTENDS FB_WorkerDefGrid IMPLEMENTS I_PrintSubsystem
VAR_INPUT
  nPrintPos             : DINT;   // Absolute printing position [SubPx]
  fMasterSpeed          : LREAL;  // Current Speed [m/s]
  bHardwareSync         : BOOL;   // hw sync signal (chenerates a triger internally)
  bHardwareHold         : BOOL;   // hw hold signal (and fast print stop request)
  bFastStopRequest      : BOOL;   // Fast stop print request
  bPrintStopRequest     : BOOL;   // Normal synchronized print stop
  fPrintStartOffset     : LREAL;  // [m] X-Shift - StartOffset from CT Detection X0 to Print (configurative PU/PM/PG/PA ADS offset + DetectToPrintDist) [m]
  fPrintYOffset         : LREAL;  // [m] Y-Shift
  nPhDepth              : UDINT;  // [px] ph depth
  // correction live parameter
  fPUElevation          : LREAL;  // PU distance from substrate [m]
END_VAR
VAR_OUTPUT
  bPrintActive          : BOOL;   // A print is activated / started
END_VAR
VAR
  // print
  // - references
  _pAdsPg            : POINTER TO FB_ADS_PG;      // pg ads reference (for pa)
  _pAdsCam           : POINTER TO ST_ADS_CAMERA;  // camera interface PUC

  // - instances
  fbPs               : FB_PS_PrintBuffer;
  fbPa               : FB_PA;
  fB_PcAdapter       : FB_PC_Adapter;
  
  // grid specific
  // - references
  _iParamMediator    : I_ParamMediator;
  // - settings
  sDefGridSettings   : ST_DefGridSettings; 

  // print corrections
  nPointCorrections  : UDINT;     // number of registered point correction handler
  iPointCorrections  : ARRAY[1..nC_NUM_POINTCORRECTIONS] OF I_GridPointCorrection;  // point corrections
  
  // - Time of flight correction of droplets
  fbDropSpeedComp    : FB_DropSpeedComp;
  bShowDropSpeedSetup : BOOL;

  // settings or helper (global or last attached ct)
  _bWorkerPrintEnable: BOOL;    // print on worker enabled 
  _nPosX0            : DINT;    // X0 for last attached CT (detected postion)
  _nPosXS            : DINT;    // XS for last attached CT (shifted print start position)
  _nPosXDelta        : DINT;    // Shift value X0 -> XS
  _fPosY             : LREAL;   // Y shift for last attached CT
  _fCurrentImgDepth  : LREAL;   // Job: current image length [m]
  _bEndless          : BOOL;    // Job: endless
  _bPaStarted        : BOOL;
  _bPaStartRequested : BOOL;
  _bPaStopping       : BOOL;
  _sJobDef           : BOOL;
  PaStartTimeout     : TON;
  rTrigHwSync        : R_TRIG;
  _bForceDefGridOff  : BOOL;    // force deformation grid stream to ph off (send 0)
  bBuffStopBit : BOOL;
  
  // grid settings
  _iPhGrid           : I_Correction_Grid;
  _sPhGridHwCfg      : ST_GridHwCfg;
  // grid limit
  _fLimitCorrectionX : LREAL;     // correction limit in y (abs) [px]
  _fLimitCorrectionY : LREAL;     // correction limit in y (abs) [px]
  _bGridWasLimited : BOOL;        // streamed grid was limited
    
  // Messaging
  (*we could implement a message handler for ST_ADS_PG message interface*)

  // History
  sRepeatHistory : ARRAY[0..nC_HistorySize-1] OF ST_RepeatHistory;
  nRepeatCt : UDINT;

  // testing
  bEnVerbose : BOOL;
END_VAR
VAR PERSISTENT
  _fColumnsToPrecharge : LREAL := nC_COLUMNS_TO_PRECHARGE;
  _fStartShiftOffset   : LREAL := fC_START_SHIFT_OFFSET;
  _fStartShiftFactor   : LREAL := fC_START_SHIFT_FACTOR;
END_VAR
VAR CONSTANT
  iC_NUM_MSG               : UDINT := 5;
  nC_COLUMNS_TO_PRECHARGE  : LREAL := 2.1;
  fC_GRIDPOINT_STREAM_TIME : LREAL := 0.0025;    // time to stream one point [s]
  fC_START_SHIFT_FACTOR    : LREAL := -0.031;   //-2.4E-2;
  fC_START_SHIFT_OFFSET    : LREAL := -0.01;    //-1.0E-2;
  nC_NUM_POINTCORRECTIONS  : UDINT := 5;
  nC_HistorySize           : UDINT := 30;
END_VAR

(*
DOC:
What will be different to FB_WorkerDefGrid_Print of DMAX
- Re-Sync StartPosDetect interface with optional camera data (y-shift)
  Clear with Attach(), security clearance
- (maybe not needed) Stream grid faster to PC (we have no break for switching the CT in endless)
- New PDI StartPostion update (+print start only for first CT) --> send to NIOS or hw buffer
- PDI GridPoint stream
- New PDI PrintingLength update (after last streamed point)
- Other rules for Worker position calculation
*)

PROPERTY aPaState : STRING
GET
aPaState := fbPa.aPaState;
END_GET
END_PROPERTY

METHOD PROTECTED  Attach : BOOL
VAR_INPUT
  iCT              : I_CT;                         (*container at triggered event position*)
END_VAR
VAR
  i : UDINT;
  bCheckErr : BOOL;
  bDeformErr : BOOL;
  eDeformStep : E_DeformationStep;
END_VAR
Attach:=FALSE;

IF NOT SUPER^.Attach(iCT:=iCT) THEN
  RETURN;
END_IF

// Additional worker checks
IF _pNewAttached = 0 THEN RETURN; END_IF

// - Additional worker checks
bDeformErr := _pNewAttached^.getDeformationStatus(eDStep=>eDeformStep);   // get latest status 

  // - job is valid?
IF _pNewAttached^.pJob = 0 OR NOT _bJobActive THEN
  LogLvl(Lvl:=E_LogSeverity.Debug, Msg:='Release: no job active');
  Release(iCT:=iCT);
  RETURN;   // do not print

// CT valid & CT present
ELSIF NOT _pNewAttached^.bValid OR NOT _pNewAttached^.bProductPresent THEN
  LogLvl(Lvl:=E_LogSeverity.Debug, Msg:='Release: no produt or not valid');
  Release(iCT:=iCT);
  RETURN;   // do not print

// Ignore start due to hardware hold  
ELSIF bHardwareHold THEN
  _pNewAttached^.AbortDeformation(sReason:=EC_Print.ecPaAbortHold.Desc, Src:=_pEcSrc^, bHideLog:=TRUE);
  Release(iCT:=iCT);
  RETURN;   // do not print

// ignore new start when stop is requested
ELSIF bPrintStopRequest OR bFastStopRequest THEN
  LogLvl(Lvl:=E_LogSeverity.Debug, Msg:='Release: stop requested');
  Release(iCT:=iCT);
  RETURN;   // do not print

// - deformation started? and no deformation error so far
ELSIF bDeformErr OR eDeformStep < E_DeformationStep.cameraStarted THEN
  Release(iCT:=iCT);  // nothing to do anymore
  
// - OK attach
ELSE
  Attach := TRUE;
END_IF


// ------------------
// NOTE: we have multi-attach, take care with editing Worker globals! 


// Prepare and Start print ---------------
// - Grid udpate settings (set in WorkerDeformation during JobStart)
sDefGridSettings := _iParamMediator.sDeformationGridSettings; 

// - clear handling data 
//    done in SUPER.Attach()  push

// - Calc print positions
//  > X Position ---
_nPosX0 := _pNewAttached^.nPosPrint_X0;         // X0 "print" position for CT (should be updated to the local position domain, not the one of CTM)
_nPosXDelta :=   F_MeterToSubPixel(fPrintStartOffset, _fPrintResolution*_fSubPxResolution)                      // + PU/PM/PG shifts
               - F_MeterToSubPixel(fbDropSpeedComp.fDropPlacementError, _fPrintResolution*_fSubPxResolution);   // - drop compensation 
_nPosXS := _nPosX0 + _nPosXDelta;   // XS effective print start position
//  > Y Position ---
//   y position (with or whithout applied global y shift from correction grid)
_fPosY :=   F_MeterToSubPixel(fPosMeter:=fPrintYOffset, fResoSubPx:=_fPrintResolution);

// error checks on position
bCheckErr := checkPrintposTiming(nStartPos:=_nPosXS, nCurrentPos:=nPrintPos);
bCheckErr := checkGridTiming(nPosXS:=_nPosXS, nPosNow:=nPrintPos);

// - Globals
fB_PcAdapter.setPrintStartPos(nX0:=_nPosXS);
fB_PcAdapter.setPrintYShift(nYShift:=FC_LREAL_TO_DINT(_fPosY));
// - Per PS (PHs)
fbPs.bPrintEnable := iCT.bValid AND iCT.bProductPresent;              // ps enables
fbPs.setGrid(sGrid:=sDefGridSettings);                                // apply correction grid settings
fbPs.setupObject(                                                     // setup print data object
  nObjId:=TO_UDINT(iCT.pCT^.iId),               // (NOTE: must be a unique id per production)
  nCopy:=1,                                     // 
  bStop:=bBuffStopBit,                          // stop after printed this object
  bDir:=FALSE, 
  nPrintStartPos:=_nPosXS,                      // 
  nImageSelection:=iCT.pCT^.sData.lPage,        // 
  nShiftedStartX:=0                             // function not used in this project
);

_pNewAttachedHdlData^.nXS := _nPosXS;           // save start pos to handling data (for calc stop pos if needed)

// Start print (initial prep->start or just start next object)
IF NOT fbPa.printStart() THEN
  LogError(Msg:='PA not ready to start at attach');
  Release(iCT := iCT);
ELSE
  // start / Update ok
  IF NOT _bPaStarted THEN 
    _bPaStartRequested := TRUE;
  END_IF
  Attach:=TRUE;
END_IF

